C03641=1057.884,320.062,395.291,173.371,36.234,156.810
C03642=1057.890,320.310,395.258,173.375,36.239,156.811
C03643=1057.896,320.558,395.223,173.378,36.243,156.812
C03644=1057.903,320.805,395.190,173.382,36.248,156.813
C03645=1057.909,321.053,395.155,173.385,36.252,156.814
C03646=1057.916,321.300,395.122,173.389,36.256,156.815
C03647=1057.922,321.548,395.087,173.392,36.260,156.816
C03648=1057.930,321.796,395.054,173.396,36.264,156.817
C03649=1057.935,322.043,395.020,173.399,36.269,156.818
C03650=1057.943,322.291,394.986,173.403,36.273,156.819
C03651=1057.949,322.539,394.951,173.406,36.277,156.820
C03652=1057.955,322.786,394.917,173.411,36.281,156.821
C03653=1057.962,323.034,394.883,173.414,36.285,156.822
C03654=1057.969,323.282,394.849,173.418,36.290,156.823
C03655=1057.976,323.528,394.815,173.421,36.294,156.823
C03656=1057.982,323.776,394.780,173.425,36.299,156.824
C03657=1057.988,324.024,394.746,173.429,36.303,156.825
C03658=1057.995,324.271,394.713,173.432,36.307,156.826
C03659=1058.002,324.519,394.678,173.436,36.311,156.827
C03660=1058.009,324.767,394.644,173.439,36.316,156.828
C03661=1058.016,325.014,394.609,173.443,36.320,156.829
C03662=1058.021,325.261,394.575,173.446,36.324,156.830
C03663=1058.029,325.509,394.541,173.451,36.328,156.831
C03664=1058.035,325.757,394.507,173.454,36.333,156.832
C03665=1058.043,326.004,394.472,173.458,36.337,156.833
C03666=1058.049,326.252,394.438,173.461,36.341,156.834
C03667=1058.055,326.499,394.404,173.465,36.345,156.835
C03668=1058.062,326.747,394.370,173.469,36.350,156.836
C03669=1058.069,326.994,394.335,173.472,36.355,156.837
C03670=1058.075,327.242,394.300,173.477,36.359,156.838
C03671=1058.083,327.489,394.266,173.480,36.363,156.839
C03672=1058.089,327.737,394.231,173.484,36.367,156.840
C03673=1058.095,327.985,394.197,173.487,36.372,156.841
C03674=1058.103,328.232,394.163,173.491,36.376,156.842
C03675=1058.109,328.480,394.128,173.494,36.380,156.843
C03676=1058.116,328.727,394.093,173.499,36.385,156.844
C03677=1058.123,328.975,394.060,173.503,36.389,156.845
C03678=1058.130,329.222,394.024,173.506,36.393,156.846
C03679=1058.136,329.470,393.990,173.510,36.398,156.847
C03680=1058.144,329.717,393.955,173.513,36.402,156.848
C03681=1058.150,329.965,393.921,173.518,36.407,156.849
C03682=1058.157,330.212,393.886,173.521,36.411,156.850
C03683=1058.164,330.460,393.852,173.525,36.416,156.851
C03684=1058.170,330.708,393.816,173.529,36.420,156.852
C03685=1058.177,330.955,393.781,173.532,36.424,156.853
C03686=1058.183,331.202,393.747,173.536,36.429,156.854
C03687=1058.190,331.450,393.712,173.540,36.433,156.855
C03688=1058.197,331.702,393.676,173.544,36.438,156.856
C03689=1058.204,331.954,393.641,173.548,36.442,156.857
C03690=1058.210,332.205,393.605,173.551,36.447,156.858
C03691=1058.218,332.457,393.570,173.556,36.452,156.859
C03692=1058.224,332.705,393.535,173.559,36.456,156.860
C03693=1058.231,332.952,393.500,173.563,36.461,156.861
C03694=1058.237,333.200,393.464,173.567,36.465,156.862
C03695=1058.244,333.447,393.429,173.571,36.470,156.863
C03696=1058.250,333.695,393.394,173.575,36.474,156.864
C03697=1058.257,333.943,393.359,173.578,36.479,156.865
C03698=1058.264,334.190,393.324,173.582,36.483,156.866
C03699=1058.271,334.437,393.289,173.587,36.488,156.867
C03700=1058.277,334.685,393.254,173.590,36.493,156.868
C03701=1058.284,334.932,393.219,173.594,36.497,156.869
C03702=1058.291,335.179,393.184,173.598,36.502,156.870
C03703=1058.298,335.427,393.148,173.602,36.507,156.871
C03704=1058.305,335.674,393.113,173.606,36.511,156.872
C03705=1058.311,335.921,393.078,173.609,36.516,156.873
C03706=1058.317,336.169,393.042,173.613,36.520,156.874
C03707=1058.324,336.417,393.007,173.618,36.525,156.876
C03708=1058.331,336.664,392.972,173.621,36.529,156.877
C03709=1058.338,336.911,392.936,173.625,36.534,156.878
C03710=1058.345,337.158,392.901,173.630,36.538,156.879
C03711=1058.351,337.406,392.865,173.633,36.544,156.880
C03712=1058.358,337.654,392.830,173.637,36.548,156.881
C03713=1058.365,337.901,392.795,173.641,36.553,156.882
C03714=1058.371,338.148,392.758,173.645,36.557,156.883
C03715=1058.378,338.396,392.723,173.649,36.562,156.884
C03716=1058.385,338.643,392.688,173.652,36.567,156.885
C03717=1058.392,338.890,392.653,173.657,36.571,156.886
C03718=1058.398,339.137,392.616,173.661,36.576,156.887
C03719=1058.405,339.385,392.581,173.664,36.581,156.888
C03720=1058.412,339.633,392.546,173.669,36.585,156.889
C03721=1058.418,339.880,392.509,173.673,36.591,156.891
C03722=1058.425,340.127,392.474,173.676,36.595,156.892
C03723=1058.431,340.374,392.438,173.681,36.600,156.893
C03724=1058.439,340.622,392.402,173.685,36.605,156.894
C03725=1058.446,340.869,392.366,173.688,36.609,156.895
C03726=1058.452,341.117,392.331,173.693,36.614,156.896
C03727=1058.459,341.364,392.296,173.697,36.619,156.897
C03728=1058.466,341.612,392.259,173.700,36.624,156.898
C03729=1058.473,341.859,392.223,173.705,36.628,156.899
C03730=1058.479,342.106,392.188,173.709,36.633,156.900
C03731=1058.487,342.353,392.152,173.713,36.638,156.901
C03732=1058.493,342.601,392.116,173.717,36.643,156.903
C03733=1058.500,342.848,392.080,173.721,36.648,156.904
C03734=1058.506,343.095,392.044,173.725,36.652,156.905
C03735=1058.514,343.343,392.008,173.729,36.657,156.906
C03736=1058.520,343.590,391.972,173.734,36.662,156.907
C03737=1058.527,343.837,391.936,173.738,36.667,156.908
C03738=1058.534,344.085,391.900,173.741,36.672,156.909
C03739=1058.541,344.332,391.864,173.746,36.677,156.910
C03740=1058.547,344.579,391.827,173.750,36.681,156.912
C03741=1058.554,344.827,391.791,173.754,36.686,156.913
C03742=1058.561,345.074,391.755,173.758,36.692,156.914
C03743=1058.567,345.321,391.719,173.762,36.696,156.915
C03744=1058.574,345.569,391.682,173.766,36.701,156.916
C03745=1058.581,345.816,391.646,173.770,36.706,156.917
C03746=1058.588,346.064,391.610,173.775,36.711,156.918
C03747=1058.594,346.311,391.574,173.779,36.716,156.919
C03748=1058.602,346.558,391.538,173.783,36.721,156.921
C03749=1058.608,346.805,391.501,173.787,36.726,156.922
C03750=1058.615,347.053,391.464,173.792,36.731,156.923
C03751=1058.622,347.300,391.428,173.796,36.736,156.924
C03752=1058.629,347.548,391.392,173.800,36.741,156.925
C03753=1058.636,347.795,391.355,173.804,36.746,156.927
C03754=1058.643,348.042,391.319,173.809,36.751,156.928
C03755=1058.650,348.289,391.283,173.812,36.756,156.929
C03756=1058.656,348.536,391.246,173.816,36.761,156.930
C03757=1058.663,348.784,391.209,173.821,36.766,156.931
C03758=1058.670,349.030,391.173,173.825,36.771,156.932
C03759=1058.677,349.278,391.136,173.829,36.776,156.933
C03760=1058.684,349.525,391.099,173.833,36.781,156.935
C03761=1058.691,349.773,391.063,173.838,36.786,156.936
C03762=1058.698,350.020,391.027,173.843,36.791,156.937
C03763=1058.705,350.267,390.989,173.846,36.796,156.938
C03764=1058.712,350.514,390.952,173.851,36.801,156.939
C03765=1058.718,350.762,390.916,173.855,36.806,156.941
C03766=1058.726,351.009,390.880,173.860,36.811,156.942
C03767=1058.733,351.255,390.843,173.863,36.816,156.943
C03768=1058.739,351.503,390.806,173.868,36.822,156.944
C03769=1058.746,351.750,390.769,173.872,36.827,156.945
C03770=1058.753,351.997,390.732,173.877,36.832,156.947
C03771=1058.760,352.245,390.695,173.881,36.837,156.948
C03772=1058.767,352.492,390.658,173.885,36.842,156.949
C03773=1058.774,352.739,390.621,173.889,36.848,156.950
C03774=1058.780,352.986,390.584,173.894,36.853,156.951
C03775=1058.787,353.233,390.547,173.899,36.858,156.953
C03776=1058.794,353.481,390.510,173.903,36.863,156.954
C03777=1058.801,353.728,390.473,173.907,36.868,156.955
C03778=1058.808,353.975,390.436,173.911,36.873,156.956
C03779=1058.815,354.222,390.398,173.916,36.879,156.958
C03780=1058.822,354.469,390.362,173.921,36.884,156.959
C03781=1058.829,354.716,390.324,173.924,36.889,156.960
C03782=1058.836,354.963,390.287,173.929,36.895,156.961
C03783=1058.842,355.210,390.250,173.933,36.900,156.963
C03784=1058.850,355.457,390.213,173.938,36.905,156.964
C03785=1058.857,355.705,390.175,173.943,36.910,156.965
C03786=1058.863,355.952,390.139,173.947,36.916,156.966
C03787=1058.870,356.199,390.101,173.951,36.921,156.968
C03788=1058.878,356.446,390.064,173.955,36.926,156.969
C03789=1058.885,356.693,390.026,173.960,36.931,156.970
C03790=1058.892,356.939,389.989,173.965,36.937,156.971
C03791=1058.899,357.187,389.951,173.969,36.942,156.973
C03792=1058.906,357.434,389.915,173.973,36.947,156.974
C03793=1058.913,357.681,389.877,173.978,36.952,156.975
C03794=1058.920,357.929,389.839,173.982,36.958,156.976
C03795=1058.927,358.176,389.802,173.987,36.964,156.978
C03796=1058.934,358.422,389.765,173.992,36.969,156.979
C03797=1058.941,358.669,389.727,173.996,36.974,156.980
C03798=1058.948,358.917,389.689,174.001,36.980,156.982
C03799=1058.955,359.164,389.652,174.005,36.985,156.983
C03800=1058.963,359.416,389.613,174.010,36.991,156.984
C03801=1058.970,359.668,389.575,174.014,36.996,156.986
C03802=1058.976,359.920,389.536,174.019,37.002,156.987
C03803=1058.983,360.172,389.498,174.024,37.008,156.988
C03804=1058.991,360.419,389.460,174.029,37.013,156.990
C03805=1058.998,360.666,389.422,174.033,37.019,156.991
C03806=1059.005,360.913,389.384,174.038,37.024,156.992
C03807=1059.012,361.160,389.346,174.042,37.029,156.993
C03808=1059.019,361.408,389.309,174.047,37.035,156.995
C03809=1059.026,361.655,389.271,174.051,37.040,156.996
C03810=1059.033,361.902,389.233,174.056,37.046,156.997
C03811=1059.040,362.149,389.195,174.061,37.051,156.999
C03812=1059.048,362.396,389.157,174.066,37.057,157.000
C03813=1059.054,362.643,389.119,174.070,37.062,157.001
C03814=1059.062,362.890,389.081,174.075,37.068,157.003
C03815=1059.069,363.136,389.043,174.080,37.074,157.004
C03816=1059.076,363.384,389.005,174.085,37.080,157.005
C03817=1059.083,363.631,388.967,174.088,37.085,157.007
C03818=1059.091,363.877,388.929,174.093,37.091,157.008
C03819=1059.097,364.125,388.891,174.098,37.096,157.009
C03820=1059.105,364.371,388.853,174.103,37.102,157.011
C03821=1059.111,364.618,388.814,174.107,37.108,157.012
C03822=1059.119,364.865,388.776,174.112,37.113,157.014
C03823=1059.125,365.112,388.737,174.117,37.119,157.015
C03824=1059.132,365.359,388.699,174.122,37.125,157.016
C03825=1059.140,365.606,388.661,174.127,37.131,157.018
C03826=1059.146,365.853,388.622,174.131,37.137,157.019
C03827=1059.154,366.099,388.584,174.136,37.142,157.021
C03828=1059.160,366.347,388.546,174.141,37.148,157.022
C03829=1059.168,366.593,388.508,174.146,37.154,157.023
C03830=1059.175,366.840,388.469,174.151,37.159,157.025
C03831=1059.182,367.087,388.430,174.156,37.165,157.026
C03832=1059.190,367.334,388.391,174.160,37.171,157.027
C03833=1059.197,367.581,388.352,174.165,37.177,157.029
C03834=1059.204,367.828,388.315,174.170,37.183,157.030
C03835=1059.211,368.075,388.276,174.175,37.189,157.032
C03836=1059.217,368.322,388.237,174.180,37.195,157.033
C03837=1059.225,368.568,388.199,174.184,37.200,157.035
C03838=1059.232,368.816,388.160,174.189,37.206,157.036
C03839=1059.240,369.062,388.122,174.194,37.212,157.038
C03840=1059.247,369.309,388.083,174.199,37.218,157.039
C03841=1059.254,369.556,388.044,174.203,37.224,157.040
C03842=1059.261,369.803,388.006,174.208,37.230,157.042
C03843=1059.269,370.050,387.966,174.214,37.236,157.043
C03844=1059.276,370.296,387.927,174.218,37.241,157.045
C03845=1059.283,370.543,387.889,174.223,37.247,157.046
C03846=1059.291,370.790,387.849,174.229,37.254,157.048
C03847=1059.298,371.037,387.811,174.234,37.260,157.049
C03848=1059.305,371.284,387.772,174.239,37.266,157.051
C03849=1059.312,371.531,387.733,174.244,37.272,157.052
C03850=1059.320,371.777,387.694,174.249,37.278,157.053
C03851=1059.327,372.024,387.655,174.254,37.283,157.055
C03852=1059.334,372.271,387.616,174.259,37.289,157.056
C03853=1059.342,372.518,387.577,174.264,37.296,157.058
C03854=1059.348,372.765,387.538,174.269,37.302,157.059
C03855=1059.356,373.012,387.499,174.274,37.308,157.061
C03856=1059.364,373.282,387.455,174.279,37.314,157.062
C03857=1059.372,373.553,387.413,174.284,37.321,157.064
C03858=1059.380,373.823,387.369,174.290,37.328,157.066
C03859=1059.388,374.094,387.327,174.296,37.335,157.067
C03860=1059.395,374.340,387.287,174.301,37.341,157.069
C03861=1059.403,374.587,387.247,174.306,37.347,157.071
C03862=1059.409,374.834,387.209,174.311,37.353,157.072
C03863=1059.417,375.081,387.169,174.316,37.359,157.074
C03864=1059.424,375.327,387.129,174.321,37.366,157.075
C03865=1059.431,375.574,387.090,174.326,37.372,157.077
C03866=1059.439,375.820,387.050,174.331,37.379,157.078
C03867=1059.446,376.067,387.011,174.336,37.385,157.080
C03868=1059.453,376.314,386.972,174.341,37.391,157.081
C03869=1059.460,376.560,386.932,174.347,37.397,157.083
C03870=1059.468,376.807,386.892,174.352,37.404,157.084
C03871=1059.475,377.053,386.853,174.358,37.410,157.086
C03872=1059.483,377.300,386.813,174.363,37.416,157.088
C03873=1059.490,377.547,386.773,174.368,37.422,157.089
C03874=1059.498,377.794,386.734,174.373,37.429,157.091
C03875=1059.505,378.041,386.694,174.378,37.435,157.092
C03876=1059.512,378.287,386.654,174.383,37.441,157.094
C03877=1059.520,378.534,386.614,174.389,37.448,157.095
C03878=1059.527,378.780,386.575,174.394,37.455,157.097
C03879=1059.535,379.027,386.535,174.399,37.461,157.099
C03880=1059.543,379.274,386.495,174.404,37.467,157.100
C03881=1059.550,379.520,386.456,174.410,37.474,157.102
C03882=1059.558,379.767,386.415,174.415,37.480,157.103
C03883=1059.566,380.014,386.375,174.421,37.487,157.105
C03884=1059.572,380.260,386.335,174.426,37.493,157.107
C03885=1059.580,380.507,386.295,174.431,37.499,157.108
C03886=1059.587,380.754,386.255,174.436,37.506,157.110
C03887=1059.595,381.001,386.215,174.442,37.513,157.112
C03888=1059.603,381.246,386.175,174.448,37.519,157.113
C03889=1059.610,381.494,386.134,174.453,37.526,157.115
C03890=1059.617,381.740,386.095,174.458,37.532,157.116
C03891=1059.624,381.986,386.054,174.463,37.539,157.118
C03892=1059.632,382.233,386.014,174.469,37.546,157.120
C03893=1059.640,382.480,385.973,174.475,37.553,157.122
C03894=1059.646,382.726,385.933,174.480,37.559,157.123
C03895=1059.654,382.972,385.892,174.485,37.566,157.125
C03896=1059.662,383.219,385.852,174.490,37.573,157.127
C03897=1059.669,383.466,385.811,174.496,37.579,157.128
C03898=1059.676,383.712,385.771,174.502,37.586,157.130
C03899=1059.684,383.958,385.731,174.507,37.593,157.132
C03900=1059.691,384.206,385.690,174.512,37.599,157.133
C03901=1059.699,384.452,385.650,174.518,37.606,157.135
C03902=1059.707,384.698,385.608,174.524,37.613,157.137
C03903=1059.714,384.945,385.569,174.529,37.620,157.138
C03904=1059.722,385.191,385.528,174.535,37.627,157.140
C03905=1059.729,385.438,385.487,174.541,37.633,157.142
C03906=1059.737,385.684,385.446,174.546,37.640,157.144
C03907=1059.744,385.931,385.406,174.552,37.648,157.145
C03908=1059.752,386.177,385.365,174.557,37.654,157.147
C03909=1059.760,386.424,385.325,174.563,37.661,157.149
C03910=1059.767,386.670,385.283,174.568,37.668,157.151
C03911=1059.775,386.916,385.243,174.574,37.675,157.152
C03912=1059.782,387.156,385.203,174.580,37.682,157.154
C03913=1059.790,387.396,385.163,174.585,37.688,157.156
C03914=1059.797,387.636,385.123,174.591,37.695,157.157
C03915=1059.805,387.874,385.084,174.596,37.702,157.159
C03916=1059.813,388.115,385.044,174.602,37.709,157.161
C03917=1059.820,388.353,385.004,174.608,37.716,157.163
C03918=1059.827,388.594,384.964,174.613,37.722,157.164
C03919=1059.835,388.833,384.925,174.618,37.729,157.166
C03920=1059.843,389.079,384.883,174.625,37.736,157.168
C03921=1059.851,389.326,384.842,174.630,37.743,157.170
C03922=1059.858,389.572,384.801,174.636,37.750,157.171
C03923=1059.866,389.819,384.760,174.642,37.757,157.173
C03924=1059.874,390.065,384.719,174.647,37.765,157.175
C03925=1059.882,390.312,384.677,174.653,37.772,157.177
C03926=1059.890,390.558,384.636,174.659,37.779,157.179
C03927=1059.897,390.805,384.595,174.665,37.786,157.181
C03928=1059.905,391.051,384.553,174.671,37.793,157.182
C03929=1059.913,391.297,384.512,174.677,37.801,157.184
C03930=1059.920,391.543,384.470,174.683,37.808,157.186
C03931=1059.928,391.790,384.429,174.689,37.815,157.188
C03932=1059.936,392.036,384.387,174.694,37.822,157.190
C03933=1059.944,392.283,384.346,174.700,37.830,157.192
C03934=1059.951,392.529,384.304,174.706,37.837,157.194
C03935=1059.959,392.775,384.263,174.712,37.844,157.196
C03936=1059.968,393.021,384.221,174.718,37.852,157.197
C03937=1059.975,393.267,384.179,174.724,37.859,157.199
C03938=1059.983,393.513,384.138,174.730,37.866,157.201
C03939=1059.990,393.760,384.096,174.736,37.874,157.203
C03940=1059.998,394.007,384.054,174.742,37.881,157.205
C03941=1060.006,394.253,384.012,174.749,37.889,157.207
C03942=1060.014,394.499,383.970,174.754,37.897,157.209
C03943=1060.021,394.746,383.928,174.761,37.904,157.211
C03944=1060.029,394.992,383.887,174.766,37.912,157.213
C03945=1060.037,395.238,383.845,174.773,37.919,157.215
C03946=1060.046,395.484,383.803,174.778,37.927,157.217
C03947=1060.053,395.730,383.761,174.785,37.934,157.219
C03948=1060.061,395.976,383.719,174.790,37.942,157.221
C03949=1060.069,396.223,383.677,174.797,37.950,157.223
C03950=1060.076,396.469,383.635,174.804,37.957,157.225
C03951=1060.085,396.716,383.592,174.809,37.965,157.227
C03952=1060.092,396.961,383.550,174.816,37.972,157.228
C03953=1060.100,397.208,383.508,174.822,37.980,157.231
C03954=1060.108,397.453,383.466,174.828,37.988,157.232
C03955=1060.117,397.700,383.423,174.835,37.996,157.235
C03956=1060.127,398.015,383.369,174.843,38.005,157.237
C03957=1060.136,398.330,383.315,174.851,38.015,157.240
C03958=1060.147,398.646,383.261,174.859,38.025,157.242
C03959=1060.157,398.960,383.206,174.867,38.036,157.245
C03960=1060.165,399.207,383.163,174.872,38.043,157.247
C03961=1060.172,399.453,383.121,174.879,38.051,157.249
C03962=1060.181,399.699,383.078,174.886,38.059,157.251
C03963=1060.189,399.946,383.036,174.891,38.067,157.253
C03964=1060.197,400.192,382.993,174.898,38.075,157.255
C03965=1060.205,400.438,382.951,174.905,38.083,157.257
C03966=1060.213,400.685,382.907,174.912,38.091,157.260
C03967=1060.220,400.931,382.865,174.917,38.099,157.262
C03968=1060.231,401.250,382.810,174.926,38.109,157.264
C03969=1060.242,401.569,382.754,174.935,38.120,157.267
C03970=1060.253,401.887,382.699,174.943,38.130,157.270
C03971=1060.264,402.206,382.643,174.951,38.141,157.273
C03972=1060.271,402.452,382.600,174.958,38.149,157.275
C03973=1060.280,402.699,382.557,174.965,38.157,157.277
C03974=1060.287,402.944,382.515,174.971,38.165,157.279
C03975=1060.295,403.191,382.471,174.977,38.174,157.281
C03976=1060.304,403.437,382.428,174.984,38.181,157.283
C03977=1060.312,403.683,382.385,174.991,38.190,157.286
C03978=1060.320,403.929,382.341,174.997,38.198,157.288
C03979=1060.328,404.175,382.298,175.004,38.206,157.290
C03980=1060.336,404.421,382.255,175.011,38.215,157.292
C03981=1060.345,404.668,382.212,175.017,38.223,157.294
C03982=1060.352,404.913,382.168,175.024,38.231,157.296
C03983=1060.360,405.159,382.125,175.031,38.240,157.299
C03984=1060.368,405.405,382.081,175.037,38.248,157.301
C03985=1060.377,405.651,382.038,175.044,38.257,157.303
C03986=1060.385,405.897,381.994,175.051,38.265,157.305
C03987=1060.393,406.143,381.951,175.058,38.274,157.308
C03988=1060.401,406.389,381.907,175.065,38.282,157.310
C03989=1060.409,406.636,381.863,175.072,38.291,157.312
C03990=1060.418,406.882,381.820,175.079,38.299,157.314
C03991=1060.426,407.127,381.776,175.086,38.308,157.317
C03992=1060.435,407.374,381.733,175.093,38.317,157.319
C03993=1060.443,407.620,381.688,175.099,38.325,157.321
C03994=1060.451,407.866,381.645,175.106,38.333,157.324
C03995=1060.459,408.112,381.601,175.113,38.342,157.326
C03996=1060.467,408.358,381.557,175.120,38.351,157.328
C03997=1060.475,408.604,381.513,175.127,38.360,157.331
C03998=1060.484,408.849,381.469,175.134,38.369,157.333
C03999=1060.492,409.096,381.425,175.141,38.377,157.335
C04000=1060.500,409.342,381.381,175.148,38.386,157.338
C04001=1060.509,409.587,381.337,175.155,38.395,157.340
C04002=1060.517,409.833,381.293,175.162,38.404,157.342
C04003=1060.525,410.079,381.248,175.169,38.413,157.345
C04004=1060.534,410.326,381.204,175.176,38.421,157.347
C04005=1060.543,410.571,381.161,175.184,38.430,157.350
C04006=1060.551,410.817,381.116,175.191,38.439,157.352
C04007=1060.559,411.064,381.072,175.198,38.448,157.354
C04008=1060.568,411.309,381.028,175.205,38.457,157.357
C04009=1060.576,411.555,380.984,175.213,38.466,157.359
C04010=1060.585,411.801,380.939,175.220,38.475,157.362
C04011=1060.593,412.047,380.895,175.228,38.484,157.364
C04012=1060.602,412.293,380.850,175.235,38.493,157.367
C04013=1060.611,412.538,380.805,175.242,38.502,157.369
C04014=1060.619,412.785,380.761,175.249,38.511,157.372
C04015=1060.627,413.030,380.716,175.257,38.520,157.374
C04016=1060.637,413.277,380.672,175.264,38.530,157.377
C04017=1060.645,413.522,380.628,175.271,38.538,157.379
C04018=1060.654,413.768,380.582,175.279,38.548,157.382
C04019=1060.662,414.014,380.538,175.287,38.557,157.384
C04020=1060.671,414.260,380.493,175.294,38.566,157.387
C04021=1060.679,414.505,380.448,175.301,38.576,157.389
C04022=1060.688,414.751,380.403,175.309,38.585,157.392
C04023=1060.696,414.997,380.359,175.317,38.594,157.394
C04024=1060.708,415.321,380.299,175.327,38.607,157.398
C04025=1060.719,415.646,380.240,175.337,38.620,157.401
C04026=1060.730,415.969,380.180,175.347,38.632,157.404
C04027=1060.742,416.294,380.120,175.357,38.645,157.408
C04028=1060.750,416.540,380.076,175.365,38.654,157.411
C04029=1060.759,416.785,380.031,175.372,38.663,157.413
C04030=1060.768,417.031,379.985,175.380,38.673,157.416
C04031=1060.776,417.277,379.940,175.388,38.683,157.418
C04032=1060.785,417.522,379.894,175.395,38.693,157.421
C04033=1060.794,417.768,379.849,175.403,38.702,157.424
C04034=1060.803,418.014,379.803,175.411,38.712,157.426
C04035=1060.811,418.259,379.758,175.419,38.721,157.429
C04036=1060.820,418.505,379.713,175.427,38.731,157.432
C04037=1060.829,418.751,379.667,175.435,38.741,157.434
C04038=1060.838,418.997,379.622,175.443,38.751,157.437
C04039=1060.846,419.243,379.576,175.451,38.761,157.440
C04040=1060.856,419.488,379.530,175.459,38.771,157.443
C04041=1060.865,419.734,379.484,175.467,38.780,157.445
C04042=1060.874,419.980,379.439,175.475,38.790,157.448
C04043=1060.882,420.225,379.394,175.484,38.800,157.451
C04044=1060.891,420.470,379.348,175.491,38.810,157.454
C04045=1060.900,420.716,379.302,175.499,38.820,157.456
C04046=1060.909,420.961,379.256,175.507,38.830,157.459
C04047=1060.917,421.207,379.210,175.515,38.840,157.462
C04048=1060.926,421.453,379.164,175.524,38.850,157.465
C04049=1060.936,421.698,379.117,175.532,38.860,157.468
C04050=1060.944,421.944,379.071,175.540,38.871,157.471
C04051=1060.953,422.189,379.025,175.549,38.881,157.473
C04052=1060.962,422.435,378.979,175.557,38.891,157.476
C04053=1060.971,422.681,378.933,175.565,38.901,157.479
C04054=1060.979,422.926,378.886,175.573,38.911,157.482
C04055=1060.989,423.172,378.840,175.582,38.922,157.485
C04056=1060.998,423.417,378.794,175.591,38.932,157.488
C04057=1061.007,423.663,378.747,175.598,38.942,157.491
C04058=1061.016,423.908,378.701,175.607,38.953,157.494
C04059=1061.025,424.153,378.654,175.616,38.964,157.497
C04060=1061.034,424.399,378.608,175.624,38.974,157.500
C04061=1061.043,424.645,378.561,175.633,38.984,157.502
C04062=1061.052,424.890,378.515,175.642,38.995,157.505
C04063=1061.061,425.136,378.468,175.651,39.005,157.508
C04064=1061.071,425.381,378.422,175.658,39.016,157.511
C04065=1061.080,425.626,378.374,175.667,39.026,157.514
C04066=1061.089,425.872,378.328,175.676,39.037,157.517
C04067=1061.098,426.118,378.281,175.685,39.048,157.520
C04068=1061.108,426.362,378.234,175.693,39.058,157.523
C04069=1061.116,426.608,378.187,175.702,39.069,157.526
C04070=1061.126,426.854,378.141,175.711,39.080,157.530
C04071=1061.135,427.099,378.093,175.720,39.091,157.533
C04072=1061.145,427.344,378.046,175.729,39.102,157.536
C04073=1061.154,427.589,377.999,175.738,39.113,157.539
C04074=1061.163,427.834,377.952,175.747,39.123,157.542
C04075=1061.172,428.080,377.904,175.755,39.134,157.545
C04076=1061.181,428.325,377.857,175.765,39.145,157.548
C04077=1061.191,428.571,377.810,175.774,39.156,157.551
C04078=1061.200,428.816,377.763,175.783,39.167,157.555
C04079=1061.209,429.061,377.715,175.792,39.179,157.558
C04080=1061.222,429.406,377.648,175.805,39.194,157.562
C04081=1061.236,429.750,377.582,175.818,39.210,157.567
C04082=1061.249,430.095,377.515,175.831,39.226,157.571
C04083=1061.262,430.440,377.448,175.844,39.242,157.576
C04084=1061.272,430.686,377.400,175.853,39.253,157.579
C04085=1061.281,430.931,377.352,175.862,39.264,157.582
C04086=1061.290,431.176,377.304,175.872,39.275,157.586
C04087=1061.300,431.421,377.256,175.882,39.287,157.589
C04088=1061.309,431.667,377.209,175.891,39.298,157.592
C04089=1061.318,431.911,377.160,175.900,39.310,157.596
C04090=1061.328,432.157,377.113,175.910,39.322,157.599
C04091=1061.337,432.402,377.064,175.919,39.333,157.602
C04092=1061.347,432.647,377.016,175.929,39.344,157.606
C04093=1061.357,432.892,376.968,175.939,39.356,157.609
C04094=1061.366,433.137,376.920,175.948,39.368,157.612
C04095=1061.375,433.382,376.872,175.958,39.379,157.616
C04096=1061.385,433.627,376.823,175.968,39.391,157.619
C04097=1061.395,433.872,376.775,175.978,39.403,157.623
C04098=1061.404,434.118,376.727,175.987,39.415,157.626
C04099=1061.414,434.362,376.678,175.998,39.427,157.630
C04100=1061.424,434.607,376.630,176.007,39.438,157.633
C04101=1061.434,434.852,376.581,176.017,39.450,157.637
C04102=1061.443,435.097,376.533,176.027,39.463,157.640
C04103=1061.453,435.342,376.484,176.037,39.474,157.644
C04104=1061.463,435.587,376.436,176.047,39.486,157.647
C04105=1061.473,435.832,376.387,176.057,39.498,157.651
C04106=1061.482,436.077,376.337,176.067,39.511,157.654
C04107=1061.492,436.323,376.289,176.077,39.523,157.658
C04108=1061.502,436.568,376.240,176.087,39.535,157.661
C04109=1061.512,436.813,376.192,176.098,39.547,157.665
C04110=1061.522,437.057,376.142,176.107,39.559,157.669
C04111=1061.532,437.302,376.094,176.118,39.571,157.672
C04112=1061.542,437.547,376.044,176.129,39.584,157.676
C04113=1061.552,437.792,375.996,176.139,39.596,157.679
C04114=1061.561,438.037,375.946,176.149,39.608,157.683
C04115=1061.572,438.282,375.897,176.160,39.621,157.687
C04116=1061.582,438.527,375.848,176.170,39.633,157.691
C04117=1061.591,438.771,375.798,176.181,39.646,157.694
C04118=1061.602,439.016,375.748,176.192,39.659,157.698
C04119=1061.612,439.261,375.700,176.201,39.671,157.702
C04120=1061.621,439.506,375.650,176.212,39.684,157.706
C04121=1061.632,439.751,375.600,176.223,39.696,157.709
C04122=1061.642,439.995,375.551,176.234,39.709,157.713
C04123=1061.652,440.241,375.501,176.244,39.722,157.717
C04124=1061.662,440.485,375.452,176.255,39.735,157.721
C04125=1061.672,440.730,375.401,176.266,39.747,157.725
C04126=1061.682,440.974,375.351,176.277,39.760,157.729
C04127=1061.692,441.220,375.301,176.288,39.773,157.733
C04128=1061.702,441.464,375.252,176.299,39.786,157.736
C04129=1061.713,441.708,375.202,176.310,39.799,157.740
C04130=1061.723,441.954,375.151,176.321,39.812,157.744
C04131=1061.733,442.198,375.102,176.333,39.825,157.748
C04132=1061.743,442.443,375.051,176.344,39.839,157.752
C04133=1061.754,442.687,375.001,176.355,39.852,157.756
C04134=1061.764,442.933,374.951,176.366,39.865,157.760
C04135=1061.774,443.177,374.900,176.377,39.878,157.764
C04136=1061.784,443.408,374.853,176.388,39.891,157.768
C04137=1061.794,443.637,374.805,176.399,39.903,157.772
C04138=1061.803,443.868,374.758,176.409,39.916,157.776
C04139=1061.813,444.098,374.710,176.420,39.929,157.780
C04140=1061.822,444.328,374.663,176.431,39.941,157.784
C04141=1061.832,444.559,374.614,176.441,39.954,157.787
C04142=1061.843,444.789,374.568,176.452,39.967,157.791
C04143=1061.853,445.020,374.519,176.463,39.980,157.795
C04144=1061.862,445.264,374.469,176.476,39.993,157.799
C04145=1061.873,445.509,374.418,176.487,40.007,157.804
C04146=1061.884,445.753,374.367,176.499,40.021,157.808
C04147=1061.895,445.998,374.316,176.511,40.034,157.812
C04148=1061.905,446.243,374.265,176.523,40.048,157.816
C04149=1061.916,446.487,374.214,176.534,40.062,157.821
C04150=1061.926,446.731,374.163,176.547,40.076,157.825
C04151=1061.937,446.975,374.111,176.558,40.090,157.829
C04152=1061.948,447.218,374.060,176.571,40.104,157.834
C04153=1061.958,447.462,374.010,176.583,40.118,157.838
C04154=1061.970,447.705,373.959,176.595,40.132,157.842
C04155=1061.983,447.950,373.909,176.607,40.145,157.846
C04156=1061.997,448.194,373.860,176.619,40.158,157.851
C04157=1062.011,448.438,373.812,176.632,40.171,157.855
C04158=1062.027,448.682,373.764,176.645,40.184,157.859
C04159=1062.044,448.928,373.717,176.657,40.196,157.863
C04160=1062.060,449.172,373.670,176.670,40.208,157.867
C04161=1062.079,449.418,373.624,176.683,40.220,157.870
C04162=1062.098,449.662,373.579,176.696,40.232,157.874
C04163=1062.118,449.908,373.535,176.709,40.243,157.878
C04164=1061.785,449.918,373.260,176.702,40.360,157.910
C04165=1061.764,449.672,373.305,176.689,40.349,157.906
C04166=1061.745,449.427,373.350,176.676,40.338,157.902
C04167=1061.726,449.182,373.396,176.663,40.326,157.899
C04168=1061.708,448.937,373.443,176.650,40.314,157.895
C04169=1061.693,448.692,373.490,176.638,40.301,157.891
C04170=1061.677,448.448,373.538,176.625,40.289,157.887
C04171=1061.662,448.202,373.586,176.612,40.276,157.883
C04172=1061.648,447.960,373.635,176.600,40.263,157.879
C04173=1061.635,447.715,373.685,176.587,40.249,157.874
C04174=1061.623,447.471,373.736,176.575,40.236,157.870
C04175=1061.612,447.228,373.786,176.563,40.222,157.866
C04176=1061.601,446.985,373.837,176.551,40.208,157.861
C04177=1061.591,446.741,373.889,176.539,40.194,157.857
C04178=1061.580,446.496,373.939,176.527,40.181,157.853
C04179=1061.569,446.251,373.991,176.514,40.167,157.848
C04180=1061.559,446.007,374.042,176.503,40.153,157.844
C04181=1061.548,445.762,374.092,176.490,40.139,157.840
C04182=1061.537,445.518,374.144,176.479,40.126,157.836
C04183=1061.527,445.273,374.195,176.467,40.112,157.831
C04184=1061.516,445.029,374.245,176.455,40.099,157.827
C04185=1061.507,444.808,374.291,176.444,40.086,157.824
C04186=1061.497,444.588,374.337,176.434,40.074,157.820
C04187=1061.488,444.367,374.383,176.424,40.062,157.816
C04188=1061.478,444.146,374.429,176.413,40.050,157.812
C04189=1061.469,443.926,374.474,176.403,40.038,157.809
C04190=1061.460,443.705,374.520,176.392,40.026,157.805
C04191=1061.451,443.484,374.566,176.382,40.013,157.801
C04192=1061.441,443.264,374.610,176.372,40.001,157.797
C04193=1061.431,443.019,374.661,176.361,39.988,157.794
C04194=1061.421,442.774,374.712,176.348,39.975,157.789
C04195=1061.410,442.529,374.762,176.337,39.962,157.785
C04196=1061.399,442.285,374.813,176.326,39.949,157.781
C04197=1061.389,442.040,374.862,176.315,39.936,157.777
C04198=1061.379,441.796,374.913,176.304,39.923,157.773
C04199=1061.368,441.551,374.963,176.293,39.910,157.770
C04200=1061.358,441.307,375.013,176.282,39.897,157.766
C04201=1061.348,441.061,375.063,176.271,39.884,157.762
C04202=1061.337,440.816,375.112,176.259,39.871,157.758
C04203=1061.328,440.572,375.162,176.248,39.858,157.754
C04204=1061.317,440.327,375.212,176.237,39.845,157.750
C04205=1061.308,440.083,375.262,176.227,39.833,157.746
C04206=1061.297,439.838,375.312,176.216,39.820,157.742
C04207=1061.287,439.593,375.361,176.206,39.807,157.739
C04208=1061.277,439.348,375.411,176.195,39.795,157.735
C04209=1061.267,439.104,375.461,176.184,39.782,157.731
C04210=1061.257,438.859,375.509,176.173,39.770,157.727
C04211=1061.247,438.613,375.559,176.163,39.757,157.723
C04212=1061.237,438.369,375.609,176.152,39.745,157.720
C04213=1061.227,438.125,375.658,176.141,39.732,157.716
C04214=1061.218,437.879,375.707,176.131,39.720,157.712
C04215=1061.208,437.634,375.757,176.121,39.707,157.709
C04216=1061.198,437.390,375.806,176.110,39.695,157.705
C04217=1061.187,437.144,375.855,176.100,39.683,157.701
C04218=1061.177,436.900,375.904,176.089,39.671,157.698
C04219=1061.167,436.655,375.952,176.079,39.659,157.694
C04220=1061.158,436.410,376.001,176.069,39.647,157.690
C04221=1061.148,436.165,376.051,176.058,39.634,157.687
C04222=1061.138,435.920,376.100,176.049,39.622,157.683
C04223=1061.128,435.675,376.148,176.038,39.610,157.680
C04224=1061.118,435.430,376.197,176.028,39.598,157.676
C04225=1061.109,435.185,376.245,176.018,39.587,157.673
C04226=1061.099,434.940,376.294,176.008,39.574,157.669
C04227=1061.089,434.695,376.342,175.998,39.563,157.666
C04228=1061.079,434.450,376.391,175.988,39.551,157.662
C04229=1061.070,434.205,376.439,175.979,39.539,157.659
C04230=1061.060,433.960,376.488,175.968,39.527,157.655
C04231=1061.050,433.715,376.536,175.959,39.516,157.652
C04232=1061.040,433.470,376.585,175.948,39.504,157.648
C04233=1061.031,433.225,376.634,175.939,39.492,157.645
C04234=1061.021,432.979,376.681,175.929,39.480,157.641
C04235=1061.011,432.734,376.730,175.920,39.469,157.638
C04236=1061.002,432.489,376.778,175.909,39.457,157.635
C04237=1060.992,432.244,376.826,175.900,39.446,157.631
C04238=1060.983,431.999,376.874,175.891,39.434,157.628
C04239=1060.973,431.754,376.922,175.881,39.423,157.625
C04240=1060.964,431.509,376.971,175.871,39.411,157.621
C04241=1060.954,431.263,377.018,175.862,39.400,157.618
C04242=1060.945,431.018,377.066,175.852,39.389,157.615
C04243=1060.936,430.773,377.114,175.843,39.377,157.611
C04244=1060.926,430.528,377.162,175.834,39.366,157.608
C04245=1060.913,430.182,377.230,175.820,39.350,157.604
C04246=1060.899,429.834,377.296,175.807,39.334,157.599
C04247=1060.886,429.488,377.364,175.794,39.318,157.594
C04248=1060.872,429.141,377.431,175.781,39.303,157.590
C04249=1060.863,428.896,377.479,175.772,39.292,157.587
C04250=1060.854,428.650,377.526,175.762,39.281,157.583
C04251=1060.845,428.405,377.573,175.753,39.270,157.580
C04252=1060.835,428.160,377.621,175.744,39.259,157.577
C04253=1060.826,427.915,377.668,175.735,39.248,157.574
C04254=1060.817,427.669,377.716,175.726,39.237,157.571
C04255=1060.808,427.424,377.763,175.718,39.226,157.568
C04256=1060.798,427.179,377.810,175.709,39.216,157.565
C04257=1060.789,426.934,377.857,175.700,39.204,157.562
C04258=1060.780,426.687,377.904,175.691,39.194,157.558
C04259=1060.771,426.443,377.951,175.682,39.183,157.556
C04260=1060.762,426.197,377.998,175.673,39.173,157.552
C04261=1060.752,425.951,378.044,175.664,39.162,157.549
C04262=1060.743,425.707,378.092,175.655,39.151,157.546
C04263=1060.733,425.461,378.138,175.647,39.141,157.543
C04264=1060.725,425.215,378.185,175.638,39.130,157.540
C04265=1060.716,424.970,378.231,175.629,39.120,157.537
C04266=1060.706,424.724,378.279,175.620,39.109,157.534
C04267=1060.697,424.479,378.325,175.611,39.099,157.531
C04268=1060.688,424.234,378.372,175.603,39.088,157.528
C04269=1060.679,423.988,378.418,175.595,39.078,157.526
C04270=1060.669,423.743,378.465,175.586,39.068,157.523
C04271=1060.661,423.497,378.511,175.578,39.057,157.520
C04272=1060.651,423.252,378.557,175.569,39.047,157.517
C04273=1060.643,423.006,378.604,175.560,39.037,157.514
C04274=1060.633,422.761,378.650,175.553,39.026,157.511
C04275=1060.625,422.516,378.697,175.544,39.016,157.508
C04276=1060.616,422.270,378.742,175.535,39.006,157.505
C04277=1060.607,422.025,378.789,175.527,38.995,157.502
C04278=1060.597,421.778,378.836,175.519,38.986,157.500
C04279=1060.588,421.533,378.881,175.510,38.975,157.497
C04280=1060.580,421.287,378.928,175.502,38.965,157.494
C04281=1060.571,421.042,378.974,175.494,38.955,157.491
C04282=1060.562,420.796,379.019,175.486,38.945,157.488
C04283=1060.554,420.551,379.066,175.477,38.935,157.485
C04284=1060.545,420.305,379.111,175.470,38.925,157.483
C04285=1060.535,420.060,379.157,175.461,38.915,157.480
C04286=1060.527,419.814,379.203,175.453,38.905,157.477
C04287=1060.518,419.567,379.249,175.445,38.895,157.474
C04288=1060.509,419.322,379.294,175.437,38.886,157.472
C04289=1060.500,419.077,379.340,175.429,38.876,157.469
C04290=1060.491,418.831,379.386,175.421,38.866,157.466
C04291=1060.482,418.586,379.431,175.412,38.857,157.463
C04292=1060.473,418.340,379.476,175.405,38.847,157.461
C04293=1060.465,418.094,379.523,175.396,38.837,157.458
C04294=1060.456,417.848,379.568,175.389,38.827,157.455
C04295=1060.447,417.603,379.613,175.381,38.818,157.453
C04296=1060.439,417.357,379.658,175.373,38.808,157.450
C04297=1060.430,417.111,379.704,175.365,38.798,157.447
C04298=1060.421,416.865,379.749,175.358,38.789,157.445
C04299=1060.412,416.620,379.794,175.350,38.780,157.442
C04300=1060.403,416.374,379.840,175.342,38.770,157.439
C04301=1060.392,416.048,379.900,175.332,38.757,157.436
C04302=1060.380,415.722,379.960,175.322,38.745,157.433
C04303=1060.369,415.395,380.020,175.312,38.732,157.429
C04304=1060.358,415.070,380.079,175.302,38.720,157.426
C04305=1060.349,414.824,380.125,175.293,38.710,157.423
C04306=1060.341,414.578,380.169,175.286,38.701,157.420
C04307=1060.332,414.333,380.214,175.279,38.692,157.418
C04308=1060.323,414.086,380.259,175.271,38.683,157.415
C04309=1060.315,413.841,380.304,175.263,38.673,157.413
C04310=1060.306,413.595,380.348,175.256,38.664,157.410
C04311=1060.298,413.349,380.393,175.248,38.655,157.408
C04312=1060.289,413.103,380.438,175.241,38.646,157.405
C04313=1060.280,412.857,380.483,175.234,38.636,157.403
C04314=1060.272,412.611,380.527,175.226,38.628,157.400
C04315=1060.262,412.365,380.571,175.218,38.619,157.398
C04316=1060.254,412.120,380.616,175.211,38.610,157.396
C04317=1060.246,411.874,380.661,175.204,38.600,157.393
C04318=1060.237,411.628,380.705,175.197,38.591,157.391
C04319=1060.229,411.382,380.749,175.189,38.583,157.388
C04320=1060.220,411.136,380.794,175.182,38.574,157.386
C04321=1060.212,410.890,380.838,175.175,38.565,157.383
C04322=1060.203,410.645,380.882,175.167,38.556,157.381
C04323=1060.194,410.398,380.927,175.160,38.547,157.378
C04324=1060.186,410.153,380.971,175.153,38.538,157.376
C04325=1060.177,409.907,381.015,175.145,38.530,157.374
C04326=1060.169,409.660,381.059,175.138,38.521,157.371
C04327=1060.161,409.414,381.103,175.131,38.512,157.369
C04328=1060.153,409.169,381.147,175.124,38.503,157.367
C04329=1060.144,408.923,381.191,175.117,38.494,157.364
C04330=1060.136,408.676,381.235,175.110,38.486,157.362
C04331=1060.128,408.430,381.279,175.103,38.477,157.360
C04332=1060.119,408.185,381.323,175.096,38.468,157.357
C04333=1060.111,407.939,381.367,175.089,38.459,157.355
C04334=1060.103,407.693,381.411,175.082,38.451,157.353
C04335=1060.095,407.447,381.454,175.075,38.442,157.350
C04336=1060.087,407.201,381.498,175.068,38.434,157.348
C04337=1060.077,406.954,381.542,175.061,38.425,157.346
C04338=1060.069,406.708,381.586,175.054,38.417,157.343
C04339=1060.062,406.462,381.630,175.047,38.408,157.341
C04340=1060.053,406.217,381.674,175.041,38.400,157.339
C04341=1060.045,405.970,381.717,175.033,38.391,157.336
C04342=1060.037,405.724,381.761,175.027,38.382,157.334
C04343=1060.028,405.479,381.805,175.020,38.374,157.332
C04344=1060.021,405.232,381.848,175.013,38.366,157.330
C04345=1060.012,404.986,381.891,175.006,38.358,157.328
C04346=1060.004,404.740,381.934,175.000,38.349,157.325
C04347=1059.996,404.494,381.978,174.993,38.341,157.323
C04348=1059.987,404.248,382.021,174.986,38.333,157.321
C04349=1059.980,404.003,382.065,174.980,38.324,157.319
C04350=1059.971,403.757,382.108,174.973,38.316,157.317
C04351=1059.964,403.510,382.151,174.966,38.308,157.314
C04352=1059.955,403.264,382.195,174.959,38.300,157.312
C04353=1059.947,403.017,382.237,174.953,38.291,157.310
C04354=1059.939,402.771,382.280,174.947,38.283,157.308
C04355=1059.931,402.525,382.323,174.940,38.275,157.306
C04356=1059.922,402.279,382.366,174.933,38.267,157.303
C04357=1059.912,401.958,382.423,174.925,38.256,157.301
C04358=1059.902,401.638,382.479,174.916,38.246,157.298
C04359=1059.891,401.317,382.534,174.907,38.236,157.295
C04360=1059.880,400.996,382.590,174.899,38.225,157.292
C04361=1059.872,400.751,382.633,174.892,38.217,157.290
C04362=1059.864,400.504,382.675,174.886,38.209,157.288
C04363=1059.856,400.258,382.718,174.880,38.201,157.286
C04364=1059.848,400.012,382.760,174.873,38.193,157.284
C04365=1059.840,399.766,382.804,174.867,38.185,157.282
C04366=1059.832,399.519,382.846,174.860,38.177,157.280
C04367=1059.824,399.273,382.889,174.854,38.169,157.278
C04368=1059.816,399.027,382.931,174.847,38.162,157.276
C04369=1059.808,398.781,382.974,174.841,38.154,157.274
C04370=1059.800,398.535,383.016,174.835,38.146,157.272
C04371=1059.793,398.288,383.059,174.828,38.138,157.270
C04372=1059.784,398.042,383.102,174.822,38.131,157.268
C04373=1059.776,397.796,383.144,174.816,38.123,157.266
C04374=1059.768,397.550,383.186,174.809,38.115,157.264
C04375=1059.760,397.304,383.229,174.803,38.107,157.261
C04376=1059.752,397.057,383.271,174.797,38.100,157.260
C04377=1059.745,396.812,383.313,174.791,38.092,157.258
C04378=1059.736,396.565,383.355,174.785,38.085,157.256
C04379=1059.729,396.319,383.397,174.778,38.077,157.254
C04380=1059.721,396.072,383.440,174.772,38.069,157.252
C04381=1059.713,395.826,383.481,174.766,38.062,157.250
C04382=1059.705,395.580,383.524,174.760,38.054,157.248
C04383=1059.696,395.334,383.565,174.754,38.047,157.246
C04384=1059.689,395.088,383.607,174.747,38.039,157.244
C04385=1059.681,394.841,383.649,174.742,38.032,157.242
C04386=1059.673,394.595,383.691,174.735,38.024,157.240
C04387=1059.665,394.349,383.733,174.730,38.017,157.238
C04388=1059.657,394.103,383.776,174.723,38.009,157.236
C04389=1059.650,393.856,383.817,174.717,38.002,157.234
C04390=1059.642,393.610,383.859,174.711,37.994,157.232
C04391=1059.634,393.363,383.901,174.705,37.987,157.230
C04392=1059.626,393.118,383.942,174.699,37.979,157.228
C04393=1059.619,392.871,383.984,174.693,37.972,157.226
C04394=1059.611,392.625,384.026,174.687,37.965,157.225
C04395=1059.603,392.378,384.068,174.681,37.958,157.223
C04396=1059.595,392.132,384.109,174.675,37.950,157.221
C04397=1059.587,391.886,384.151,174.669,37.943,157.219
C04398=1059.580,391.640,384.192,174.663,37.936,157.217
C04399=1059.572,391.393,384.234,174.657,37.928,157.215
C04400=1059.564,391.147,384.275,174.651,37.921,157.213
C04401=1059.556,390.901,384.317,174.646,37.914,157.211
C04402=1059.549,390.654,384.358,174.639,37.907,157.210
C04403=1059.540,390.408,384.399,174.634,37.900,157.208
C04404=1059.533,390.162,384.440,174.627,37.893,157.206
C04405=1059.526,389.915,384.482,174.622,37.885,157.204
C04406=1059.517,389.668,384.523,174.616,37.878,157.202
C04407=1059.510,389.422,384.565,174.610,37.871,157.200
C04408=1059.502,389.176,384.605,174.604,37.864,157.199
C04409=1059.494,388.929,384.646,174.598,37.857,157.197
C04410=1059.486,388.683,384.687,174.593,37.850,157.195
C04411=1059.479,388.437,384.728,174.587,37.843,157.193
C04412=1059.471,388.190,384.769,174.581,37.836,157.191
C04413=1059.461,387.886,384.820,174.574,37.827,157.189
C04414=1059.452,387.583,384.871,174.566,37.819,157.187
C04415=1059.442,387.280,384.920,174.560,37.810,157.185
C04416=1059.432,386.977,384.971,174.553,37.802,157.183
C04417=1059.425,386.730,385.012,174.547,37.795,157.181
C04418=1059.417,386.483,385.052,174.541,37.788,157.179
C04419=1059.409,386.237,385.093,174.536,37.781,157.177
C04420=1059.402,385.990,385.134,174.530,37.774,157.176
C04421=1059.394,385.744,385.175,174.524,37.767,157.174
C04422=1059.387,385.497,385.216,174.519,37.760,157.172
C04423=1059.379,385.251,385.257,174.514,37.754,157.171
C04424=1059.372,385.004,385.297,174.507,37.747,157.169
C04425=1059.362,384.716,385.344,174.501,37.739,157.167
C04426=1059.353,384.426,385.392,174.494,37.731,157.165
C04427=1059.344,384.138,385.440,174.488,37.723,157.163
C04428=1059.336,383.849,385.487,174.481,37.715,157.161
C04429=1059.329,383.602,385.528,174.476,37.708,157.159
C04430=1059.321,383.356,385.569,174.471,37.702,157.157
C04431=1059.313,383.109,385.609,174.466,37.695,157.156
C04432=1059.306,382.863,385.650,174.459,37.688,157.154
C04433=1059.299,382.616,385.689,174.454,37.682,157.152
C04434=1059.291,382.370,385.731,174.449,37.675,157.151
C04435=1059.284,382.123,385.771,174.443,37.669,157.149
C04436=1059.276,381.877,385.811,174.438,37.662,157.147
C04437=1059.269,381.630,385.851,174.432,37.655,157.146
C04438=1059.261,381.383,385.891,174.427,37.649,157.144
C04439=1059.254,381.138,385.932,174.421,37.642,157.142
C04440=1059.247,380.890,385.972,174.416,37.636,157.141
C04441=1059.239,380.643,386.012,174.411,37.629,157.139
C04442=1059.232,380.397,386.052,174.406,37.623,157.137
C04443=1059.224,380.151,386.092,174.400,37.616,157.136
C04444=1059.216,379.904,386.132,174.394,37.609,157.134
C04445=1059.209,379.657,386.172,174.389,37.603,157.133
C04446=1059.202,379.411,386.212,174.384,37.596,157.131
C04447=1059.194,379.164,386.251,174.379,37.590,157.129
C04448=1059.186,378.917,386.291,174.374,37.584,157.128
C04449=1059.179,378.671,386.331,174.368,37.577,157.126
C04450=1059.171,378.424,386.371,174.362,37.571,157.125
C04451=1059.164,378.177,386.411,174.357,37.565,157.123
C04452=1059.156,377.931,386.450,174.352,37.558,157.121
C04453=1059.150,377.684,386.491,174.347,37.552,157.120
C04454=1059.142,377.438,386.530,174.341,37.546,157.118
C04455=1059.135,377.191,386.570,174.336,37.539,157.117
C04456=1059.128,376.944,386.610,174.331,37.533,157.115
C04457=1059.120,376.698,386.650,174.326,37.527,157.114
C04458=1059.112,376.450,386.689,174.321,37.521,157.112
C04459=1059.105,376.204,386.729,174.316,37.514,157.110
C04460=1059.098,375.957,386.768,174.311,37.508,157.109
C04461=1059.090,375.711,386.808,174.305,37.502,157.107
C04462=1059.082,375.463,386.847,174.300,37.495,157.106
C04463=1059.075,375.217,386.886,174.295,37.489,157.104
C04464=1059.068,374.971,386.926,174.290,37.483,157.103
C04465=1059.061,374.733,386.964,174.285,37.477,157.101
C04466=1059.054,374.494,387.003,174.280,37.471,157.100
C04467=1059.047,374.255,387.040,174.275,37.465,157.098
C04468=1059.040,374.017,387.078,174.270,37.459,157.097
C04469=1059.033,373.779,387.116,174.265,37.453,157.095
C04470=1059.026,373.541,387.154,174.260,37.447,157.094
C04471=1059.019,373.303,387.192,174.256,37.441,157.092
C04472=1059.012,373.065,387.231,174.251,37.436,157.091
C04473=1059.005,372.817,387.270,174.245,37.429,157.089
C04474=1058.998,372.570,387.309,174.240,37.423,157.088
C04475=1058.991,372.324,387.348,174.235,37.417,157.086
C04476=1058.983,372.077,387.387,174.230,37.411,157.085
C04477=1058.976,371.831,387.426,174.225,37.405,157.083
C04478=1058.969,371.584,387.465,174.220,37.399,157.082
C04479=1058.961,371.337,387.504,174.215,37.393,157.081
C04480=1058.954,371.090,387.543,174.210,37.388,157.079
C04481=1058.947,370.844,387.582,174.205,37.381,157.078
C04482=1058.939,370.596,387.621,174.200,37.375,157.076
C04483=1058.932,370.350,387.660,174.195,37.369,157.075
C04484=1058.925,370.103,387.698,174.190,37.363,157.073
C04485=1058.917,369.856,387.737,174.185,37.358,157.072
C04486=1058.910,369.609,387.776,174.180,37.352,157.070
C04487=1058.903,369.362,387.814,174.176,37.346,157.069
C04488=1058.896,369.115,387.853,174.171,37.340,157.068
C04489=1058.888,368.868,387.892,174.166,37.334,157.066
C04490=1058.881,368.621,387.930,174.161,37.328,157.065
C04491=1058.874,368.375,387.969,174.156,37.323,157.063
C04492=1058.867,368.128,388.008,174.151,37.317,157.062
C04493=1058.860,367.881,388.046,174.146,37.311,157.060
C04494=1058.852,367.634,388.086,174.141,37.305,157.059
C04495=1058.845,367.387,388.124,174.137,37.299,157.058
C04496=1058.838,367.140,388.163,174.132,37.293,157.056
C04497=1058.830,366.894,388.201,174.127,37.287,157.055
C04498=1058.823,366.647,388.240,174.122,37.282,157.053
C04499=1058.817,366.400,388.278,174.117,37.276,157.052
C04500=1058.809,366.153,388.316,174.112,37.270,157.051
C04501=1058.803,365.906,388.355,174.108,37.265,157.049
C04502=1058.795,365.660,388.393,174.103,37.259,157.048
C04503=1058.788,365.412,388.432,174.098,37.253,157.046
C04504=1058.781,365.165,388.470,174.093,37.248,157.045
C04505=1058.774,364.918,388.509,174.088,37.242,157.044
C04506=1058.767,364.671,388.547,174.084,37.236,157.042
C04507=1058.759,364.424,388.585,174.079,37.231,157.041
C04508=1058.753,364.177,388.624,174.074,37.224,157.039
C04509=1058.745,363.930,388.661,174.069,37.219,157.038
C04510=1058.739,363.684,388.700,174.064,37.213,157.037
C04511=1058.731,363.436,388.738,174.060,37.208,157.035
C04512=1058.724,363.190,388.776,174.055,37.202,157.034
C04513=1058.717,362.942,388.814,174.050,37.197,157.033
C04514=1058.710,362.696,388.852,174.045,37.191,157.031
C04515=1058.703,362.449,388.890,174.041,37.186,157.030
C04516=1058.696,362.201,388.928,174.036,37.180,157.029
C04517=1058.688,361.955,388.966,174.032,37.175,157.027
C04518=1058.681,361.708,389.004,174.027,37.169,157.026
C04519=1058.675,361.460,389.042,174.023,37.164,157.025
C04520=1058.667,361.214,389.080,174.018,37.158,157.023
C04521=1058.660,360.967,389.118,174.013,37.152,157.022
C04522=1058.653,360.719,389.155,174.008,37.147,157.021
C04523=1058.647,360.473,389.193,174.004,37.141,157.019
C04524=1058.639,360.226,389.231,173.999,37.136,157.018
C04525=1058.632,359.971,389.270,173.994,37.130,157.017
C04526=1058.625,359.718,389.309,173.989,37.125,157.015
C04527=1058.617,359.465,389.347,173.985,37.119,157.014
C04528=1058.610,359.210,389.386,173.981,37.114,157.013
C04529=1058.603,358.963,389.423,173.976,37.108,157.011
C04530=1058.596,358.716,389.461,173.971,37.103,157.010
C04531=1058.589,358.469,389.499,173.967,37.098,157.009
C04532=1058.582,358.222,389.536,173.962,37.092,157.008
C04533=1058.575,357.974,389.574,173.957,37.086,157.006
C04534=1058.568,357.728,389.611,173.953,37.081,157.005
C04535=1058.561,357.481,389.648,173.948,37.076,157.004
C04536=1058.554,357.234,389.686,173.944,37.071,157.003
C04537=1058.546,356.987,389.724,173.940,37.065,157.001
C04538=1058.540,356.739,389.762,173.935,37.060,157.000
C04539=1058.533,356.493,389.799,173.930,37.055,156.999
C04540=1058.526,356.246,389.836,173.926,37.050,156.997
C04541=1058.519,355.998,389.873,173.921,37.044,156.996
C04542=1058.512,355.751,389.911,173.918,37.039,156.995
C04543=1058.505,355.504,389.948,173.913,37.034,156.994
C04544=1058.498,355.257,389.985,173.908,37.029,156.992
C04545=1058.491,355.009,390.022,173.904,37.023,156.991
C04546=1058.484,354.762,390.060,173.899,37.018,156.990
C04547=1058.477,354.516,390.097,173.895,37.013,156.989
C04548=1058.470,354.268,390.134,173.890,37.007,156.987
C04549=1058.463,354.021,390.171,173.886,37.002,156.986
C04550=1058.456,353.774,390.208,173.882,36.997,156.985
C04551=1058.449,353.527,390.245,173.877,36.992,156.984
C04552=1058.442,353.280,390.283,173.873,36.987,156.983
C04553=1058.436,353.033,390.319,173.868,36.982,156.981
C04554=1058.428,352.785,390.357,173.864,36.976,156.980
C04555=1058.422,352.538,390.393,173.860,36.971,156.979
C04556=1058.415,352.291,390.431,173.855,36.966,156.978
C04557=1058.407,352.044,390.467,173.851,36.961,156.976
C04558=1058.400,351.797,390.504,173.846,36.956,156.975
C04559=1058.394,351.550,390.541,173.843,36.950,156.974
C04560=1058.387,351.303,390.578,173.838,36.945,156.973
C04561=1058.380,351.055,390.615,173.834,36.940,156.972
C04562=1058.373,350.808,390.652,173.829,36.935,156.970
C04563=1058.367,350.561,390.688,173.825,36.930,156.969
C04564=1058.359,350.314,390.725,173.821,36.925,156.968
C04565=1058.352,350.067,390.761,173.817,36.920,156.967
C04566=1058.345,349.819,390.798,173.812,36.915,156.966
C04567=1058.339,349.572,390.835,173.808,36.910,156.964
C04568=1058.331,349.325,390.872,173.804,36.905,156.963
C04569=1058.325,349.078,390.908,173.800,36.900,156.962
C04570=1058.318,348.830,390.945,173.795,36.895,156.961
C04571=1058.310,348.583,390.981,173.791,36.890,156.960
C04572=1058.304,348.336,391.018,173.786,36.885,156.959
C04573=1058.298,348.089,391.054,173.783,36.880,156.957
C04574=1058.290,347.842,391.092,173.778,36.875,156.956
C04575=1058.283,347.595,391.127,173.774,36.870,156.955
C04576=1058.276,347.347,391.164,173.769,36.865,156.954
C04577=1058.270,347.100,391.201,173.766,36.860,156.953
C04578=1058.262,346.853,391.237,173.761,36.855,156.952
C04579=1058.256,346.606,391.273,173.757,36.850,156.950
C04580=1058.249,346.358,391.310,173.753,36.846,156.949
C04581=1058.242,346.109,391.346,173.749,36.841,156.948
C04582=1058.235,345.860,391.382,173.744,36.836,156.947
C04583=1058.229,345.610,391.419,173.740,36.830,156.946
C04584=1058.222,345.361,391.455,173.735,36.825,156.945
C04585=1058.215,345.114,391.492,173.732,36.821,156.944
C04586=1058.208,344.867,391.528,173.728,36.816,156.942
C04587=1058.201,344.620,391.565,173.723,36.811,156.941
C04588=1058.194,344.373,391.600,173.720,36.806,156.940
C04589=1058.188,344.124,391.637,173.715,36.801,156.939
C04590=1058.181,343.877,391.673,173.711,36.796,156.938
C04591=1058.174,343.631,391.709,173.707,36.792,156.937
C04592=1058.167,343.383,391.746,173.703,36.787,156.936
C04593=1058.161,343.136,391.781,173.699,36.782,156.935
C04594=1058.154,342.888,391.817,173.694,36.777,156.933
C04595=1058.147,342.641,391.853,173.691,36.772,156.932
C04596=1058.140,342.393,391.889,173.687,36.767,156.931
C04597=1058.133,342.147,391.925,173.682,36.763,156.930
C04598=1058.126,341.899,391.960,173.678,36.758,156.929
C04599=1058.120,341.651,391.997,173.675,36.753,156.928
C04600=1058.113,341.404,392.032,173.670,36.748,156.927
C04601=1058.106,341.157,392.068,173.666,36.744,156.926
C04602=1058.099,340.909,392.104,173.662,36.739,156.925
C04603=1058.092,340.662,392.140,173.658,36.734,156.923
C04604=1058.085,340.415,392.175,173.654,36.730,156.922
C04605=1058.079,340.168,392.211,173.650,36.725,156.921
C04606=1058.072,339.920,392.247,173.646,36.720,156.920
C04607=1058.065,339.673,392.283,173.642,36.716,156.919
C04608=1058.059,339.425,392.319,173.638,36.710,156.918
C04609=1058.052,339.178,392.354,173.634,36.706,156.917
C04610=1058.045,338.931,392.390,173.630,36.701,156.916
C04611=1058.038,338.683,392.426,173.626,36.697,156.915
C04612=1058.031,338.435,392.461,173.622,36.692,156.914
C04613=1058.025,338.188,392.497,173.618,36.687,156.913
C04614=1058.018,337.941,392.532,173.615,36.683,156.912
C04615=1058.011,337.694,392.567,173.610,36.678,156.910
C04616=1058.005,337.446,392.603,173.606,36.673,156.909
C04617=1057.998,337.199,392.639,173.603,36.669,156.908
C04618=1057.992,336.952,392.674,173.598,36.664,156.907
C04619=1057.985,336.705,392.709,173.594,36.660,156.906
C04620=1057.977,336.456,392.745,173.591,36.654,156.905
C04621=1057.971,336.209,392.781,173.587,36.650,156.904
C04622=1057.965,335.961,392.816,173.582,36.645,156.903
C04623=1057.958,335.714,392.851,173.579,36.641,156.902
C04624=1057.951,335.467,392.886,173.575,36.636,156.901
C04625=1057.944,335.219,392.921,173.570,36.632,156.900
C04626=1057.938,334.972,392.956,173.567,36.627,156.899
C04627=1057.931,334.725,392.991,173.563,36.623,156.898
C04628=1057.924,334.477,393.026,173.560,36.618,156.897
C04629=1057.917,334.230,393.062,173.555,36.614,156.896
C04630=1057.911,333.983,393.097,173.551,36.609,156.895
C04631=1057.904,333.735,393.132,173.548,36.605,156.894
C04632=1057.898,333.488,393.168,173.544,36.600,156.893
C04633=1057.891,333.240,393.203,173.540,36.595,156.892
C04634=1057.884,332.993,393.238,173.536,36.591,156.891
C04635=1057.877,332.745,393.273,173.532,36.586,156.889
C04636=1057.871,332.498,393.308,173.528,36.582,156.888
C04637=1057.864,332.244,393.343,173.525,36.577,156.887
C04638=1057.856,331.991,393.379,173.520,36.573,156.886
C04639=1057.850,331.738,393.416,173.517,36.568,156.885
C04640=1057.843,331.483,393.451,173.513,36.564,156.884
C04641=1057.836,331.236,393.486,173.509,36.559,156.883
C04642=1057.830,330.989,393.521,173.505,36.555,156.882
C04643=1057.823,330.741,393.556,173.501,36.550,156.881
C04644=1057.817,330.494,393.590,173.497,36.545,156.880
C04645=1057.810,330.247,393.626,173.494,36.541,156.879
C04646=1057.804,329.999,393.660,173.490,36.537,156.878
C04647=1057.796,329.752,393.695,173.486,36.532,156.877
C04648=1057.790,329.504,393.729,173.482,36.528,156.876
C04649=1057.783,329.256,393.764,173.479,36.524,156.875
C04650=1057.776,329.009,393.798,173.475,36.519,156.874
C04651=1057.769,328.761,393.833,173.471,36.515,156.873
C04652=1057.763,328.513,393.867,173.468,36.511,156.872
C04653=1057.755,328.266,393.902,173.463,36.507,156.871
C04654=1057.749,328.018,393.936,173.460,36.502,156.870
C04655=1057.742,327.771,393.972,173.456,36.498,156.869
C04656=1057.735,327.523,394.005,173.452,36.494,156.868
C04657=1057.728,327.276,394.041,173.449,36.489,156.867
C04658=1057.722,327.029,394.075,173.445,36.485,156.866
C04659=1057.715,326.781,394.108,173.441,36.480,156.865
C04660=1057.708,326.534,394.144,173.437,36.476,156.865
C04661=1057.702,326.286,394.178,173.434,36.472,156.864
C04662=1057.694,326.038,394.212,173.430,36.468,156.863
C04663=1057.688,325.790,394.247,173.426,36.463,156.862
C04664=1057.682,325.543,394.281,173.423,36.459,156.861
C04665=1057.675,325.296,394.315,173.419,36.455,156.860
C04666=1057.668,325.048,394.349,173.416,36.451,156.859
C04667=1057.661,324.801,394.384,173.412,36.446,156.858
C04668=1057.655,324.553,394.418,173.408,36.442,156.857
C04669=1057.648,324.305,394.452,173.404,36.438,156.856
C04670=1057.641,324.058,394.486,173.401,36.434,156.855
C04671=1057.635,323.810,394.520,173.397,36.429,156.854
C04672=1057.628,323.563,394.555,173.393,36.425,156.853
C04673=1057.621,323.315,394.589,173.390,36.420,156.852
C04674=1057.615,323.067,394.624,173.386,36.416,156.851
C04675=1057.608,322.820,394.657,173.383,36.412,156.850
C04676=1057.602,322.572,394.691,173.379,36.408,156.849
C04677=1057.595,322.325,394.725,173.376,36.404,156.848
C04678=1057.589,322.077,394.759,173.372,36.399,156.847
C04679=1057.581,321.830,394.793,173.369,36.395,156.846
C04680=1057.575,321.582,394.828,173.365,36.391,156.845
C04681=1057.569,321.334,394.862,173.361,36.387,156.844
C04682=1057.562,321.087,394.895,173.358,36.383,156.844
C04683=1057.555,320.839,394.930,173.353,36.378,156.842
C04684=1057.549,320.592,394.963,173.350,36.374,156.842
C04685=1057.542,320.344,394.998,173.346,36.370,156.841
C04686=1057.536,320.097,395.031,173.343,36.365,156.840
C04687=1057.529,319.849,395.066,173.339,36.361,156.839
C04688=1057.522,319.601,395.099,173.336,36.357,156.838
C04689=1057.516,319.354,395.133,173.332,36.353,156.837
C04690=1057.509,319.106,395.167,173.329,36.349,156.836
C04691=1057.504,318.858,395.201,173.325,36.344,156.835
C04692=1057.496,318.611,395.234,173.321,36.340,156.834
C04693=1057.490,318.352,395.270,173.318,36.336,156.833
C04694=1057.483,318.093,395.305,173.314,36.332,156.832
C04695=1057.477,317.834,395.341,173.311,36.327,156.831
C04696=1057.470,317.575,395.377,173.307,36.323,156.830
C04697=1057.464,317.327,395.409,173.304,36.318,156.829
C04698=1057.457,317.079,395.444,173.300,36.314,156.828
C04699=1057.451,316.832,395.477,173.297,36.310,156.827
C04700=1057.445,316.585,395.511,173.293,36.306,156.827
C04701=1057.438,316.337,395.544,173.290,36.302,156.825
C04702=1057.432,316.090,395.578,173.286,36.298,156.825
C04703=1057.425,315.842,395.612,173.283,36.294,156.824
C04704=1057.418,315.594,395.645,173.279,36.290,156.823
C04705=1057.412,315.346,395.679,173.276,36.285,156.822
C04706=1057.406,315.099,395.712,173.272,36.281,156.821
C04707=1057.400,314.852,395.746,173.269,36.277,156.820
C04708=1057.393,314.604,395.780,173.266,36.273,156.819
C04709=1057.387,314.356,395.813,173.262,36.268,156.818
C04710=1057.380,314.109,395.847,173.259,36.264,156.817
C04711=1057.374,313.860,395.880,173.255,36.260,156.816
C04712=1057.368,313.613,395.914,173.252,36.256,156.815
C04713=1057.361,313.366,395.947,173.248,36.252,156.815
C04714=1057.355,313.117,395.980,173.245,36.248,156.814
C04715=1057.348,312.871,396.013,173.241,36.244,156.813
C04716=1057.341,312.622,396.046,173.238,36.240,156.812
C04717=1057.335,312.375,396.079,173.234,36.236,156.811
C04718=1057.328,312.127,396.113,173.231,36.232,156.810
C04719=1057.321,311.879,396.146,173.227,36.228,156.809
C04720=1057.314,311.631,396.179,173.224,36.224,156.808
C04721=1057.308,311.384,396.212,173.221,36.220,156.808
C04722=1057.301,311.137,396.245,173.217,36.216,156.807
C04723=1057.295,310.888,396.278,173.215,36.212,156.806
C04724=1057.288,310.641,396.311,173.211,36.208,156.805
C04725=1057.281,310.392,396.344,173.208,36.204,156.804
C04726=1057.275,310.145,396.377,173.204,36.200,156.803
C04727=1057.269,309.898,396.410,173.201,36.196,156.802
C04728=1057.262,309.649,396.443,173.197,36.192,156.801
C04729=1057.255,309.402,396.475,173.194,36.189,156.801
C04730=1057.248,309.155,396.508,173.190,36.185,156.800
C04731=1057.242,308.907,396.541,173.187,36.181,156.799
C04732=1057.235,308.659,396.574,173.183,36.177,156.798
C04733=1057.228,308.412,396.607,173.181,36.173,156.797
C04734=1057.222,308.164,396.640,173.177,36.168,156.796
C04735=1057.215,307.916,396.673,173.174,36.165,156.795
C04736=1057.209,307.668,396.706,173.170,36.161,156.794
C04737=1057.203,307.421,396.739,173.167,36.157,156.794
C04738=1057.196,307.173,396.771,173.163,36.153,156.793
C04739=1057.189,306.925,396.804,173.160,36.149,156.792
C04740=1057.183,306.677,396.837,173.157,36.145,156.791
C04741=1057.176,306.430,396.870,173.154,36.141,156.790
C04742=1057.170,306.182,396.902,173.151,36.137,156.789
C04743=1057.164,305.935,396.935,173.147,36.133,156.788
C04744=1057.157,305.687,396.968,173.144,36.129,156.788
C04745=1057.151,305.438,397.000,173.140,36.126,156.787
C04746=1057.144,305.191,397.032,173.137,36.122,156.786
C04747=1057.137,304.943,397.065,173.134,36.117,156.785
C04748=1057.131,304.696,397.098,173.131,36.113,156.784
C04749=1057.125,304.440,397.132,173.127,36.109,156.783
C04750=1057.118,304.186,397.165,173.124,36.105,156.782
C04751=1057.111,303.931,397.199,173.120,36.101,156.781
C04752=1057.105,303.677,397.232,173.117,36.097,156.781
C04753=1057.099,303.429,397.264,173.114,36.094,156.780
C04754=1057.093,303.181,397.297,173.111,36.090,156.779
C04755=1057.085,302.933,397.329,173.108,36.086,156.778
C04756=1057.079,302.686,397.362,173.104,36.082,156.777
C04757=1057.073,302.438,397.394,173.101,36.078,156.776
C04758=1057.066,302.190,397.427,173.098,36.074,156.776
C04759=1057.060,301.942,397.460,173.095,36.070,156.775
C04760=1057.054,301.694,397.492,173.091,36.066,156.774
C04761=1057.047,301.447,397.524,173.088,36.062,156.773
C04762=1057.041,301.199,397.557,173.084,36.058,156.772
C04763=1057.035,300.951,397.589,173.082,36.054,156.771
C04764=1057.028,300.703,397.621,173.079,36.050,156.770
C04765=1057.022,300.456,397.654,173.075,36.047,156.770
C04766=1057.015,300.208,397.685,173.072,36.043,156.769
C04767=1057.009,299.960,397.718,173.069,36.039,156.768
C04768=1057.003,299.712,397.750,173.066,36.035,156.767
C04769=1056.997,299.465,397.783,173.062,36.031,156.766
C04770=1056.990,299.217,397.814,173.060,36.027,156.765
C04771=1056.984,298.969,397.847,173.056,36.023,156.765
C04772=1056.978,298.721,397.879,173.053,36.019,156.764
C04773=1056.972,298.473,397.912,173.050,36.015,156.763
C04774=1056.966,298.225,397.944,173.047,36.011,156.762
C04775=1056.959,297.978,397.976,173.044,36.008,156.761
C04776=1056.953,297.730,398.008,173.040,36.004,156.760
C04777=1056.947,297.483,398.040,173.038,36.000,156.759
C04778=1056.941,297.234,398.073,173.034,35.996,156.759
C04779=1056.934,296.987,398.104,173.031,35.992,156.758
C04780=1056.928,296.739,398.137,173.028,35.988,156.757
C04781=1056.922,296.491,398.169,173.025,35.984,156.756
C04782=1056.915,296.243,398.200,173.022,35.980,156.755
C04783=1056.909,295.995,398.233,173.018,35.977,156.755
C04784=1056.902,295.747,398.264,173.016,35.973,156.754
C04785=1056.896,295.499,398.296,173.012,35.969,156.753
C04786=1056.889,295.251,398.328,173.009,35.965,156.752
C04787=1056.884,295.004,398.360,173.007,35.962,156.751
C04788=1056.877,294.756,398.392,173.003,35.958,156.750
C04789=1056.870,294.509,398.423,173.000,35.954,156.750
C04790=1056.864,294.260,398.455,172.997,35.950,156.749
C04791=1056.858,294.012,398.486,172.994,35.946,156.748
C04792=1056.852,293.764,398.519,172.990,35.942,156.747
C04793=1056.845,293.517,398.551,172.987,35.939,156.746
C04794=1056.838,293.269,398.582,172.985,35.935,156.746
C04795=1056.832,293.021,398.614,172.981,35.931,156.745
C04796=1056.825,292.773,398.646,172.978,35.927,156.744
C04797=1056.819,292.526,398.677,172.975,35.924,156.743
C04798=1056.813,292.277,398.709,172.972,35.920,156.742
C04799=1056.806,292.030,398.740,172.970,35.916,156.742
C04800=1056.800,291.782,398.772,172.966,35.913,156.741
C04801=1056.794,291.538,398.802,172.963,35.908,156.740
C04802=1056.788,291.294,398.833,172.960,35.905,156.739
C04803=1056.781,291.051,398.864,172.957,35.901,156.738
C04804=1056.775,290.807,398.896,172.955,35.897,156.738
C04805=1056.769,290.564,398.926,172.951,35.894,156.737
C04806=1056.762,290.321,398.957,172.948,35.890,156.736
C04807=1056.756,290.077,398.988,172.945,35.887,156.735
C04808=1056.750,289.834,399.019,172.942,35.883,156.734
C04809=1056.743,289.586,399.051,172.940,35.879,156.734
C04810=1056.737,289.338,399.082,172.936,35.876,156.733
C04811=1056.731,289.091,399.113,172.933,35.872,156.732
C04812=1056.724,288.842,399.144,172.930,35.868,156.731
C04813=1056.718,288.594,399.176,172.927,35.864,156.730
C04814=1056.711,288.346,399.207,172.925,35.860,156.730
C04815=1056.705,288.099,399.238,172.921,35.857,156.729
C04816=1056.699,287.851,399.270,172.918,35.853,156.728
C04817=1056.692,287.602,399.301,172.916,35.849,156.727
C04818=1056.685,287.354,399.332,172.912,35.846,156.727
C04819=1056.679,287.107,399.363,172.910,35.842,156.726
C04820=1056.673,286.859,399.394,172.906,35.838,156.725
C04821=1056.667,286.610,399.426,172.903,35.835,156.724
C04822=1056.660,286.363,399.457,172.901,35.831,156.723
C04823=1056.654,286.115,399.488,172.897,35.827,156.723
C04824=1056.648,285.867,399.519,172.895,35.824,156.722
C04825=1056.641,285.619,399.550,172.891,35.820,156.721
C04826=1056.635,285.370,399.581,172.888,35.816,156.720
C04827=1056.628,285.123,399.612,172.886,35.812,156.720
C04828=1056.622,284.875,399.643,172.882,35.809,156.719
C04829=1056.615,284.627,399.674,172.880,35.805,156.718
C04830=1056.609,284.379,399.705,172.876,35.801,156.717
C04831=1056.603,284.131,399.736,172.874,35.798,156.716
C04832=1056.596,283.883,399.767,172.871,35.794,156.716
C04833=1056.590,283.635,399.798,172.868,35.791,156.715
C04834=1056.584,283.387,399.829,172.865,35.787,156.714
C04835=1056.577,283.139,399.860,172.862,35.783,156.713
C04836=1056.571,282.891,399.890,172.859,35.779,156.713
C04837=1056.564,282.643,399.922,172.856,35.775,156.712
C04838=1056.559,282.395,399.952,172.853,35.772,156.711
C04839=1056.552,282.147,399.984,172.850,35.768,156.710
C04840=1056.546,281.899,400.014,172.848,35.765,156.709
C04841=1056.540,281.651,400.045,172.844,35.761,156.709
C04842=1056.533,281.403,400.076,172.842,35.757,156.708
C04843=1056.527,281.155,400.107,172.839,35.754,156.707
C04844=1056.520,280.907,400.138,172.836,35.750,156.706
C04845=1056.515,280.660,400.168,172.833,35.746,156.706
C04846=1056.508,280.411,400.199,172.830,35.742,156.705
C04847=1056.501,280.163,400.230,172.827,35.739,156.704
C04848=1056.496,279.915,400.261,172.825,35.735,156.703
C04849=1056.489,279.667,400.292,172.821,35.731,156.702
C04850=1056.483,279.419,400.322,172.819,35.728,156.702
C04851=1056.476,279.171,400.352,172.816,35.724,156.701
C04852=1056.470,278.924,400.383,172.813,35.721,156.700
C04853=1056.464,278.675,400.414,172.810,35.717,156.699
C04854=1056.457,278.427,400.445,172.808,35.713,156.699
C04855=1056.451,278.179,400.474,172.804,35.709,156.698
C04856=1056.444,277.931,400.505,172.802,35.706,156.697
C04857=1056.439,277.693,400.534,172.798,35.702,156.696
C04858=1056.432,277.455,400.563,172.796,35.699,156.696
C04859=1056.426,277.217,400.593,172.794,35.695,156.695
C04860=1056.420,276.979,400.622,172.790,35.692,156.694
C04861=1056.414,276.742,400.651,172.788,35.688,156.693
C04862=1056.408,276.503,400.680,172.786,35.685,156.693
C04863=1056.403,276.264,400.710,172.782,35.682,156.692
C04864=1056.396,276.027,400.740,172.780,35.678,156.691
C04865=1056.390,275.779,400.769,172.777,35.675,156.691
C04866=1056.383,275.531,400.800,172.774,35.670,156.690
C04867=1056.377,275.283,400.830,172.772,35.667,156.689
C04868=1056.370,275.035,400.861,172.769,35.663,156.688
C04869=1056.364,274.787,400.891,172.766,35.660,156.687
C04870=1056.359,274.539,400.921,172.763,35.656,156.687
C04871=1056.351,274.291,400.951,172.761,35.653,156.686
C04872=1056.346,274.043,400.982,172.757,35.649,156.685
C04873=1056.339,273.794,401.012,172.755,35.645,156.684
C04874=1056.333,273.546,401.041,172.753,35.642,156.684
C04875=1056.326,273.298,401.072,172.749,35.638,156.683
C04876=1056.321,273.050,401.103,172.747,35.634,156.682
C04877=1056.314,272.802,401.132,172.744,35.631,156.681
C04878=1056.308,272.554,401.163,172.741,35.627,156.681
C04879=1056.301,272.306,401.193,172.738,35.624,156.680
C04880=1056.295,272.057,401.223,172.736,35.620,156.679
C04881=1056.288,271.810,401.252,172.733,35.616,156.678
C04882=1056.282,271.561,401.283,172.730,35.613,156.678
C04883=1056.276,271.313,401.314,172.727,35.609,156.677
C04884=1056.270,271.065,401.343,172.724,35.605,156.676
C04885=1056.264,270.817,401.373,172.722,35.602,156.675
C04886=1056.257,270.569,401.403,172.719,35.598,156.675
C04887=1056.251,270.321,401.433,172.716,35.595,156.674
C04888=1056.244,270.073,401.463,172.714,35.591,156.673
C04889=1056.238,269.825,401.493,172.710,35.588,156.672
C04890=1056.231,269.577,401.523,172.708,35.584,156.672
C04891=1056.225,269.328,401.552,172.706,35.581,156.671
C04892=1056.219,269.081,401.583,172.702,35.577,156.670
C04893=1056.212,268.832,401.612,172.700,35.573,156.669
C04894=1056.207,268.584,401.642,172.698,35.569,156.669
C04895=1056.200,268.336,401.672,172.694,35.566,156.668
C04896=1056.194,268.087,401.702,172.692,35.562,156.667
C04897=1056.187,267.840,401.732,172.689,35.559,156.666
C04898=1056.181,267.592,401.761,172.686,35.555,156.666
C04899=1056.175,267.343,401.792,172.684,35.552,156.665
C04900=1056.168,267.095,401.821,172.681,35.548,156.664
C04901=1056.162,266.847,401.851,172.678,35.544,156.664
C04902=1056.156,266.599,401.880,172.676,35.541,156.663
C04903=1056.149,266.351,401.910,172.673,35.537,156.662
C04904=1056.143,266.103,401.939,172.670,35.534,156.661
C04905=1056.137,265.855,401.970,172.668,35.530,156.661
C04906=1056.130,265.606,401.999,172.665,35.527,156.660
C04907=1056.124,265.358,402.028,172.662,35.523,156.659
C04908=1056.118,265.110,402.058,172.660,35.520,156.658
C04909=1056.112,264.862,402.088,172.657,35.516,156.658
C04910=1056.105,264.614,402.118,172.654,35.512,156.657
C04911=1056.099,264.365,402.147,172.652,35.509,156.656
C04912=1056.093,264.117,402.176,172.649,35.505,156.655
C04913=1056.087,263.881,402.205,172.646,35.502,156.655
C04914=1056.081,263.645,402.233,172.644,35.498,156.654
C04915=1056.074,263.409,402.261,172.642,35.495,156.653
C04916=1056.069,263.174,402.289,172.640,35.492,156.653
C04917=1056.063,262.937,402.316,172.636,35.488,156.652
C04918=1056.057,262.701,402.345,172.634,35.485,156.651
C04919=1056.051,262.465,402.373,172.632,35.482,156.651
C04920=1056.045,262.229,402.401,172.629,35.478,156.650
C04921=1056.039,261.981,402.430,172.626,35.474,156.649
C04922=1056.032,261.732,402.459,172.624,35.471,156.648
C04923=1056.025,261.484,402.488,172.621,35.467,156.648
C04924=1056.019,261.236,402.518,172.619,35.464,156.647
C04925=1056.013,260.988,402.547,172.616,35.461,156.646
C04926=1056.005,260.739,402.575,172.613,35.457,156.646
C04927=1055.999,260.492,402.605,172.611,35.454,156.645
C04928=1055.993,260.244,402.634,172.608,35.450,156.644
C04929=1055.986,259.996,402.663,172.606,35.446,156.643
C04930=1055.979,259.747,402.693,172.603,35.443,156.643
C04931=1055.973,259.499,402.722,172.601,35.439,156.642
C04932=1055.967,259.251,402.751,172.598,35.436,156.641
C04933=1055.961,259.002,402.780,172.595,35.432,156.640
C04934=1055.954,258.754,402.809,172.593,35.429,156.640
C04935=1055.948,258.506,402.838,172.590,35.425,156.639
C04936=1055.941,258.257,402.867,172.587,35.422,156.638
C04937=1055.935,258.009,402.896,172.585,35.419,156.638
C04938=1055.929,257.761,402.925,172.583,35.415,156.637
C04939=1055.923,257.513,402.954,172.579,35.411,156.636
C04940=1055.916,257.265,402.983,172.577,35.408,156.635
C04941=1055.910,257.017,403.012,172.575,35.404,156.635
C04942=1055.904,256.769,403.041,172.573,35.401,156.634
C04943=1055.897,256.520,403.071,172.569,35.397,156.633
C04944=1055.890,256.271,403.099,172.567,35.394,156.633
C04945=1055.884,256.023,403.128,172.565,35.390,156.632
C04946=1055.878,255.775,403.157,172.562,35.386,156.631
C04947=1055.872,255.527,403.186,172.559,35.383,156.630
C04948=1055.865,255.279,403.215,172.557,35.379,156.630
C04949=1055.859,255.031,403.244,172.554,35.376,156.629
C04950=1055.853,254.782,403.273,172.552,35.372,156.628
C04951=1055.847,254.534,403.301,172.550,35.368,156.627
C04952=1055.841,254.286,403.330,172.546,35.365,156.627
C04953=1055.834,254.037,403.359,172.544,35.361,156.626
C04954=1055.827,253.790,403.388,172.542,35.358,156.625
C04955=1055.821,253.541,403.416,172.540,35.354,156.624
C04956=1055.815,253.293,403.445,172.537,35.351,156.624
C04957=1055.809,253.045,403.474,172.534,35.347,156.623
C04958=1055.803,252.796,403.503,172.532,35.343,156.622
C04959=1055.797,252.548,403.531,172.529,35.340,156.622
C04960=1055.791,252.300,403.560,172.527,35.336,156.621
C04961=1055.784,252.051,403.590,172.525,35.333,156.620
C04962=1055.778,251.803,403.618,172.521,35.329,156.619
C04963=1055.771,251.555,403.646,172.519,35.326,156.619
C04964=1055.765,251.307,403.675,172.517,35.322,156.618
C04965=1055.759,251.058,403.704,172.515,35.318,156.617
C04966=1055.753,250.810,403.733,172.512,35.315,156.616
C04967=1055.747,250.562,403.762,172.510,35.311,156.616
C04968=1055.741,250.313,403.790,172.508,35.308,156.615
C04969=1055.734,250.077,403.817,172.504,35.305,156.614
C04970=1055.728,249.839,403.845,172.502,35.301,156.614
C04971=1055.723,249.602,403.872,172.500,35.297,156.613
C04972=1055.717,249.365,403.900,172.497,35.294,156.612
C04973=1055.711,249.129,403.927,172.495,35.291,156.612
C04974=1055.705,248.891,403.954,172.493,35.287,156.611
C04975=1055.699,248.654,403.982,172.491,35.284,156.610
C04976=1055.693,248.417,404.008,172.488,35.280,156.609
C04977=1055.687,248.169,404.037,172.486,35.277,156.609
C04978=1055.681,247.920,404.065,172.484,35.273,156.608
C04979=1055.675,247.673,404.094,172.481,35.269,156.607
C04980=1055.669,247.424,404.122,172.479,35.266,156.607
C04981=1055.662,247.176,404.151,172.477,35.262,156.606
C04982=1055.656,246.927,404.179,172.474,35.259,156.605
C04983=1055.650,246.679,404.208,172.471,35.255,156.604
C04984=1055.644,246.431,404.237,172.469,35.251,156.604
C04985=1055.639,246.182,404.265,172.467,35.248,156.603
C04986=1055.632,245.935,404.293,172.464,35.244,156.602
C04987=1055.626,245.686,404.321,172.462,35.241,156.601
C04988=1055.620,245.437,404.350,172.460,35.237,156.601
C04989=1055.613,245.189,404.378,172.458,35.234,156.600
C04990=1055.607,244.941,404.406,172.455,35.230,156.599
C04991=1055.600,244.692,404.434,172.452,35.226,156.599
C04992=1055.594,244.444,404.463,172.450,35.223,156.598
C04993=1055.589,244.196,404.491,172.447,35.219,156.597
C04994=1055.582,243.948,404.519,172.445,35.216,156.596
C04995=1055.576,243.699,404.547,172.443,35.212,156.596
C04996=1055.569,243.451,404.576,172.441,35.208,156.595
C04997=1055.563,243.202,404.604,172.438,35.205,156.594
C04998=1055.556,242.954,404.632,172.436,35.201,156.593
C04999=1055.551,242.706,404.660,172.434,35.198,156.593
C05000=1055.545,242.457,404.688,172.431,35.194,156.592
C05001=1055.538,242.209,404.716,172.429,35.190,156.591
C05002=1055.532,241.960,404.745,172.427,35.187,156.591
C05003=1055.525,241.712,404.772,172.425,35.183,156.590
C05004=1055.519,241.464,404.800,172.421,35.180,156.589
C05005=1055.513,241.215,404.828,172.419,35.176,156.588
C05006=1055.507,240.967,404.856,172.417,35.172,156.588
C05007=1055.500,240.719,404.884,172.414,35.169,156.587
C05008=1055.494,240.470,404.912,172.412,35.165,156.586
C05009=1055.488,240.222,404.939,172.410,35.162,156.586
C05010=1055.482,239.973,404.968,172.408,35.159,156.585
C05011=1055.475,239.725,404.995,172.405,35.155,156.584
C05012=1055.469,239.476,405.023,172.403,35.152,156.583
C05013=1055.463,239.228,405.051,172.401,35.148,156.583
C05014=1055.457,238.980,405.079,172.399,35.144,156.582
C05015=1055.450,238.732,405.107,172.396,35.141,156.581
C05016=1055.443,238.483,405.134,172.394,35.137,156.581
C05017=1055.437,238.234,405.163,172.392,35.134,156.580
C05018=1055.431,237.987,405.190,172.389,35.130,156.579
C05019=1055.425,237.738,405.218,172.387,35.126,156.578
C05020=1055.419,237.489,405.246,172.385,35.123,156.578
C05021=1055.412,237.241,405.274,172.383,35.119,156.577
C05022=1055.406,236.993,405.301,172.380,35.116,156.576
C05023=1055.399,236.745,405.329,172.378,35.112,156.576
C05024=1055.394,236.495,405.356,172.376,35.108,156.575
C05025=1055.387,236.256,405.383,172.374,35.105,156.574
C05026=1055.381,236.016,405.410,172.371,35.102,156.573
C05027=1055.375,235.777,405.437,172.369,35.098,156.573
C05028=1055.369,235.536,405.463,172.367,35.095,156.572
C05029=1055.363,235.296,405.490,172.365,35.091,156.571
C05030=1055.357,235.056,405.517,172.362,35.088,156.571
C05031=1055.351,234.816,405.543,172.360,35.084,156.570
C05032=1055.345,234.576,405.570,172.358,35.081,156.569
C05033=1055.339,234.328,405.597,172.356,35.077,156.569
C05034=1055.333,234.079,405.626,172.353,35.074,156.568
C05035=1055.326,233.831,405.653,172.351,35.070,156.567
C05036=1055.320,233.582,405.680,172.349,35.066,156.566
C05037=1055.314,233.334,405.708,172.346,35.063,156.566
C05038=1055.308,233.086,405.736,172.344,35.059,156.565
C05039=1055.302,232.837,405.763,172.342,35.055,156.564
C05040=1055.295,232.588,405.790,172.340,35.052,156.564
C05041=1055.289,232.340,405.818,172.337,35.048,156.563
C05042=1055.283,232.091,405.845,172.335,35.045,156.562
C05043=1055.276,231.843,405.872,172.333,35.041,156.561
C05044=1055.270,231.595,405.900,172.331,35.037,156.561
C05045=1055.264,231.346,405.927,172.328,35.034,156.560
C05046=1055.258,231.098,405.955,172.326,35.030,156.559
C05047=1055.252,230.849,405.982,172.324,35.027,156.558
C05048=1055.245,230.601,406.010,172.323,35.023,156.558
C05049=1055.239,230.353,406.037,172.320,35.019,156.557
C05050=1055.233,230.104,406.064,172.318,35.016,156.556
C05051=1055.227,229.856,406.091,172.316,35.012,156.556
C05052=1055.220,229.607,406.118,172.314,35.009,156.555
C05053=1055.214,229.359,406.146,172.311,35.005,156.554
C05054=1055.208,229.110,406.173,172.309,35.001,156.553
C05055=1055.201,228.862,406.200,172.307,34.998,156.553
C05056=1055.195,228.613,406.227,172.304,34.994,156.552
C05057=1055.189,228.365,406.255,172.302,34.991,156.551
C05058=1055.183,228.117,406.281,172.300,34.987,156.551
C05059=1055.176,227.868,406.308,172.298,34.983,156.550
C05060=1055.169,227.619,406.336,172.295,34.980,156.549
C05061=1055.163,227.371,406.362,172.293,34.976,156.548
C05062=1055.157,227.123,406.390,172.291,34.973,156.548
C05063=1055.151,226.874,406.417,172.289,34.969,156.547
C05064=1055.145,226.625,406.444,172.287,34.965,156.546
C05065=1055.138,226.377,406.471,172.285,34.962,156.546
C05066=1055.132,226.128,406.498,172.283,34.959,156.545
C05067=1055.126,225.880,406.524,172.281,34.955,156.544
C05068=1055.119,225.632,406.552,172.278,34.951,156.544
C05069=1055.113,225.384,406.578,172.276,34.948,156.543
C05070=1055.107,225.134,406.605,172.274,34.944,156.542
C05071=1055.101,224.887,406.633,172.272,34.941,156.541
C05072=1055.094,224.638,406.660,172.269,34.936,156.541
C05073=1055.089,224.389,406.686,172.267,34.933,156.540
C05074=1055.081,224.141,406.713,172.265,34.929,156.539
C05075=1055.075,223.893,406.740,172.264,34.926,156.538
C05076=1055.069,223.644,406.767,172.261,34.922,156.538
C05077=1055.063,223.395,406.794,172.259,34.918,156.537
C05078=1055.057,223.146,406.821,172.257,34.915,156.536
C05079=1055.051,222.899,406.848,172.255,34.911,156.536
C05080=1055.044,222.650,406.875,172.252,34.907,156.535
C05081=1055.038,222.406,406.900,172.250,34.904,156.534
C05082=1055.032,222.162,406.927,172.249,34.900,156.533
C05083=1055.026,221.919,406.954,172.247,34.897,156.533
C05084=1055.020,221.674,406.980,172.244,34.893,156.532
C05085=1055.014,221.430,407.006,172.242,34.889,156.531
C05086=1055.007,221.187,407.033,172.240,34.886,156.531
C05087=1055.001,220.942,407.058,172.238,34.882,156.530
C05088=1054.995,220.699,407.085,172.236,34.879,156.529
C05089=1054.989,220.450,407.111,172.234,34.875,156.528
C05090=1054.983,220.201,407.138,172.232,34.871,156.528
C05091=1054.976,219.953,407.165,172.230,34.868,156.527
C05092=1054.970,219.705,407.191,172.228,34.865,156.526
C05093=1054.963,219.456,407.218,172.225,34.861,156.526
C05094=1054.958,219.208,407.244,172.224,34.857,156.525
C05095=1054.950,218.959,407.271,172.222,34.853,156.524
C05096=1054.945,218.711,407.297,172.220,34.850,156.523
C05097=1054.939,218.462,407.324,172.217,34.846,156.523
C05098=1054.932,218.214,407.350,172.215,34.842,156.522
C05099=1054.926,217.965,407.377,172.213,34.839,156.521
C05100=1054.919,217.716,407.403,172.212,34.835,156.521
C05101=1054.913,217.468,407.430,172.209,34.832,156.520
C05102=1054.907,217.220,407.456,172.207,34.828,156.519
C05103=1054.900,216.971,407.483,172.205,34.824,156.518
C05104=1054.894,216.723,407.510,172.203,34.821,156.518
C05105=1054.888,216.474,407.535,172.200,34.817,156.517
C05106=1054.882,216.225,407.562,172.199,34.813,156.516
C05107=1054.875,215.977,407.588,172.197,34.810,156.516
C05108=1054.870,215.728,407.615,172.195,34.806,156.515
C05109=1054.862,215.480,407.641,172.193,34.803,156.514
C05110=1054.857,215.231,407.668,172.190,34.799,156.513
C05111=1054.850,214.983,407.694,172.189,34.795,156.513
C05112=1054.844,214.734,407.720,172.187,34.791,156.512
C05113=1054.838,214.486,407.746,172.185,34.787,156.511
C05114=1054.832,214.237,407.773,172.182,34.784,156.510
C05115=1054.825,213.988,407.799,172.180,34.780,156.510
C05116=1054.819,213.739,407.825,172.179,34.777,156.509
C05117=1054.813,213.491,407.851,172.177,34.773,156.508
C05118=1054.807,213.243,407.878,172.174,34.769,156.508
C05119=1054.800,212.994,407.904,172.172,34.765,156.507
C05120=1054.794,212.745,407.930,172.171,34.762,156.506
C05121=1054.788,212.497,407.956,172.169,34.758,156.505
C05122=1054.782,212.249,407.983,172.166,34.754,156.505
C05123=1054.775,212.000,408.010,172.164,34.751,156.504
C05124=1054.769,211.751,408.035,172.163,34.747,156.503
C05125=1054.763,211.503,408.062,172.161,34.743,156.502
C05126=1054.756,211.255,408.088,172.159,34.740,156.502
C05127=1054.750,211.005,408.114,172.156,34.736,156.501
C05128=1054.744,210.757,408.140,172.154,34.732,156.500
C05129=1054.738,210.509,408.165,172.153,34.728,156.500
C05130=1054.732,210.260,408.192,172.151,34.725,156.499
C05131=1054.725,210.012,408.218,172.148,34.721,156.498
C05132=1054.719,209.763,408.244,172.146,34.717,156.497
C05133=1054.713,209.515,408.270,172.145,34.714,156.497
C05134=1054.707,209.266,408.296,172.143,34.710,156.496
C05135=1054.699,209.017,408.322,172.140,34.706,156.495
C05136=1054.694,208.768,408.348,172.138,34.702,156.494
C05137=1054.688,208.528,408.373,172.137,34.699,156.494
C05138=1054.682,208.286,408.398,172.135,34.695,156.493
C05139=1054.675,208.045,408.423,172.133,34.691,156.492
C05140=1054.669,207.804,408.448,172.131,34.688,156.492
C05141=1054.663,207.562,408.474,172.129,34.684,156.491
C05142=1054.657,207.321,408.498,172.127,34.681,156.490
C05143=1054.651,207.080,408.524,172.126,34.678,156.490
C05144=1054.644,206.838,408.549,172.124,34.674,156.489
C05145=1054.619,205.787,408.655,171.916,34.582,156.474
C05146=1054.614,205.539,408.679,171.914,34.579,156.474
C05147=1054.607,205.290,408.704,171.911,34.576,156.473
C05148=1054.602,205.041,408.729,171.908,34.573,156.473
C05149=1054.596,204.793,408.754,171.906,34.571,156.472
C05150=1054.590,204.544,408.779,171.904,34.567,156.472
C05151=1054.584,204.295,408.804,171.901,34.564,156.471
C05152=1054.577,204.047,408.828,171.899,34.562,156.471
C05153=1054.572,203.798,408.853,171.897,34.559,156.470
C05154=1054.565,203.549,408.878,171.895,34.556,156.470
C05155=1054.560,203.301,408.902,171.891,34.553,156.469
C05156=1054.554,203.052,408.928,171.889,34.550,156.468
C05157=1054.548,202.803,408.952,171.887,34.548,156.468
C05158=1054.542,202.555,408.977,171.884,34.544,156.467
C05159=1054.536,202.305,409.002,171.882,34.542,156.467
C05160=1054.530,202.057,409.027,171.880,34.539,156.466
C05161=1054.524,201.809,409.051,171.878,34.536,156.466
C05162=1054.518,201.559,409.075,171.874,34.533,156.465
C05163=1054.512,201.311,409.101,171.872,34.530,156.465
C05164=1054.506,201.062,409.124,171.870,34.528,156.464
C05165=1054.500,200.813,409.149,171.868,34.525,156.464
C05166=1054.493,200.565,409.174,171.865,34.522,156.463
C05167=1054.488,200.316,409.198,171.863,34.519,156.463
C05168=1054.482,200.067,409.223,171.861,34.516,156.462
C05169=1054.475,199.818,409.247,171.858,34.514,156.462
C05170=1054.470,199.570,409.272,171.855,34.511,156.461
C05171=1054.463,199.321,409.296,171.853,34.508,156.461
C05172=1054.457,199.072,409.321,171.851,34.506,156.460
C05173=1054.451,198.824,409.345,171.849,34.503,156.460
C05174=1054.445,198.575,409.369,171.846,34.500,156.459
C05175=1054.440,198.326,409.394,171.844,34.497,156.459
C05176=1054.433,198.077,409.418,171.842,34.495,156.458
C05177=1054.427,197.828,409.443,171.839,34.492,156.458
C05178=1054.421,197.580,409.467,171.836,34.489,156.457
C05179=1054.415,197.331,409.491,171.834,34.486,156.457
C05180=1054.409,197.083,409.515,171.832,34.483,156.456
C05181=1054.403,196.833,409.540,171.830,34.481,156.456
C05182=1054.397,196.586,409.564,171.827,34.478,156.455
C05183=1054.391,196.336,409.589,171.825,34.475,156.455
C05184=1054.385,196.087,409.613,171.823,34.473,156.454
C05185=1054.379,195.839,409.637,171.820,34.470,156.454
C05186=1054.373,195.589,409.661,171.818,34.467,156.453
C05187=1054.367,195.341,409.685,171.815,34.465,156.453
C05188=1054.361,195.092,409.710,171.813,34.461,156.452
C05189=1054.355,194.844,409.733,171.811,34.459,156.452
C05190=1054.349,194.594,409.758,171.809,34.456,156.451
C05191=1054.343,194.347,409.782,171.807,34.453,156.451
C05192=1054.337,194.097,409.807,171.803,34.451,156.450
C05193=1054.331,193.849,409.831,171.801,34.448,156.450
C05194=1054.325,193.600,409.855,171.799,34.445,156.449
C05195=1054.319,193.352,409.879,171.797,34.443,156.449
C05196=1054.313,193.102,409.904,171.795,34.440,156.448
C05197=1054.307,192.854,409.927,171.793,34.437,156.448
C05198=1054.301,192.605,409.952,171.790,34.435,156.447
C05199=1054.295,192.356,409.976,171.788,34.431,156.447
C05200=1054.290,192.108,410.000,171.785,34.429,156.446
C05201=1054.283,191.859,410.024,171.783,34.426,156.446
C05202=1054.278,191.610,410.048,171.781,34.423,156.445
C05203=1054.271,191.361,410.071,171.778,34.421,156.445
C05204=1054.266,191.112,410.096,171.776,34.418,156.444
C05205=1054.259,190.863,410.120,171.774,34.415,156.444
C05206=1054.253,190.580,410.147,171.772,34.412,156.443
C05207=1054.246,190.295,410.174,171.769,34.409,156.442
C05208=1054.240,190.012,410.203,171.766,34.406,156.442
C05209=1054.233,189.727,410.230,171.763,34.403,156.441
C05210=1054.227,189.478,410.254,171.761,34.400,156.441
C05211=1054.221,189.230,410.277,171.759,34.398,156.440
C05212=1054.215,188.981,410.302,171.757,34.395,156.440
C05213=1054.209,188.732,410.325,171.755,34.392,156.439
C05214=1054.204,188.483,410.350,171.753,34.390,156.439
C05215=1054.197,188.234,410.373,171.751,34.387,156.438
C05216=1054.192,187.986,410.397,171.747,34.384,156.438
C05217=1054.186,187.737,410.421,171.745,34.381,156.437
C05218=1054.181,187.488,410.445,171.743,34.379,156.437
C05219=1054.175,187.239,410.469,171.741,34.376,156.436
C05220=1054.169,186.990,410.493,171.739,34.373,156.436
C05221=1054.163,186.742,410.517,171.737,34.371,156.436
C05222=1054.158,186.493,410.541,171.735,34.368,156.435
C05223=1054.152,186.244,410.564,171.733,34.365,156.434
C05224=1054.145,185.995,410.588,171.731,34.363,156.434
C05225=1054.140,185.746,410.612,171.727,34.360,156.433
C05226=1054.134,185.498,410.635,171.725,34.357,156.433
C05227=1054.128,185.249,410.660,171.723,34.354,156.433
C05228=1054.122,185.000,410.684,171.721,34.352,156.432
C05229=1054.117,184.751,410.707,171.719,34.349,156.432
C05230=1054.111,184.503,410.731,171.717,34.346,156.431
C05231=1054.105,184.253,410.754,171.715,34.344,156.431
C05232=1054.099,184.005,410.778,171.713,34.341,156.430
C05233=1054.093,183.757,410.802,171.710,34.339,156.430
C05234=1054.086,183.507,410.825,171.708,34.336,156.429
C05235=1054.080,183.259,410.848,171.705,34.334,156.429
C05236=1054.074,183.009,410.872,171.703,34.331,156.428
C05237=1054.068,182.761,410.895,171.701,34.329,156.428
C05238=1054.062,182.512,410.918,171.699,34.326,156.427
C05239=1054.055,182.263,410.942,171.697,34.323,156.427
C05240=1054.050,182.014,410.965,171.695,34.321,156.426
C05241=1054.044,181.765,410.988,171.693,34.318,156.426
C05242=1054.037,181.516,411.012,171.691,34.316,156.426
C05243=1054.032,181.267,411.035,171.688,34.313,156.425
C05244=1054.026,181.019,411.059,171.685,34.310,156.425
C05245=1054.019,180.770,411.082,171.683,34.308,156.424
C05246=1054.013,180.521,411.106,171.681,34.306,156.424
C05247=1054.007,180.273,411.128,171.679,34.304,156.423
C05248=1054.001,180.024,411.151,171.677,34.301,156.423
C05249=1053.994,179.775,411.175,171.675,34.299,156.422
C05250=1053.989,179.526,411.198,171.673,34.296,156.422
C05251=1053.983,179.277,411.221,171.671,34.293,156.422
C05252=1053.976,179.028,411.245,171.669,34.291,156.421
C05253=1053.971,178.779,411.268,171.666,34.288,156.421
C05254=1053.965,178.530,411.291,171.664,34.286,156.420
C05255=1053.959,178.282,411.315,171.662,34.283,156.420
C05256=1053.952,178.032,411.338,171.659,34.281,156.419
C05257=1053.946,177.784,411.360,171.657,34.278,156.419
C05258=1053.940,177.535,411.384,171.655,34.276,156.418
C05259=1053.934,177.287,411.407,171.653,34.273,156.418
C05260=1053.928,177.037,411.430,171.651,34.271,156.418
C05261=1053.922,176.788,411.453,171.649,34.268,156.417
C05262=1053.916,176.540,411.477,171.647,34.266,156.417
C05263=1053.910,176.291,411.500,171.644,34.263,156.416
C05264=1053.905,176.042,411.523,171.642,34.261,156.416
C05265=1053.898,175.793,411.546,171.640,34.258,156.415
C05266=1053.891,175.544,411.569,171.638,34.256,156.415
C05267=1053.886,175.296,411.592,171.636,34.253,156.414
C05268=1053.880,175.047,411.615,171.634,34.251,156.414
C05269=1053.874,174.798,411.638,171.632,34.248,156.413
C05270=1053.867,174.513,411.665,171.630,34.245,156.413
C05271=1053.860,174.228,411.691,171.627,34.242,156.412
C05272=1053.853,173.944,411.717,171.625,34.239,156.412
C05273=1053.847,173.660,411.744,171.622,34.237,156.411
C05274=1053.841,173.411,411.766,171.620,34.234,156.411
C05275=1053.835,173.162,411.789,171.618,34.232,156.411
C05276=1053.829,172.913,411.812,171.616,34.229,156.410
C05277=1053.823,172.664,411.835,171.614,34.227,156.410
C05278=1053.817,172.415,411.858,171.612,34.224,156.409
C05279=1053.811,172.166,411.881,171.610,34.222,156.409
C05280=1053.805,171.918,411.904,171.608,34.219,156.408
C05281=1053.799,171.669,411.926,171.606,34.217,156.408
C05282=1053.793,171.420,411.950,171.604,34.214,156.407
C05283=1053.787,171.171,411.973,171.601,34.212,156.407
C05284=1053.782,170.923,411.996,171.599,34.209,156.406
C05285=1053.776,170.674,412.019,171.597,34.206,156.406
C05286=1053.769,170.424,412.042,171.595,34.204,156.406
C05287=1053.763,170.175,412.065,171.593,34.201,156.405
C05288=1053.757,169.927,412.088,171.591,34.199,156.405
C05289=1053.752,169.678,412.111,171.589,34.196,156.404
C05290=1053.746,169.429,412.133,171.587,34.194,156.404
C05291=1053.739,169.180,412.156,171.585,34.191,156.403
C05292=1053.734,168.931,412.178,171.583,34.189,156.403
C05293=1053.728,168.682,412.201,171.581,34.186,156.402
C05294=1053.723,168.433,412.224,171.578,34.184,156.402
C05295=1053.717,168.184,412.247,171.576,34.181,156.402
C05296=1053.710,167.935,412.269,171.574,34.179,156.401
C05297=1053.705,167.686,412.292,171.572,34.176,156.401
C05298=1053.699,167.438,412.315,171.570,34.174,156.400
C05299=1053.693,167.189,412.338,171.568,34.172,156.400
C05300=1053.687,166.940,412.361,171.566,34.169,156.399
C05301=1053.681,166.691,412.383,171.564,34.167,156.399
C05302=1053.676,166.442,412.406,171.562,34.164,156.398
C05303=1053.670,166.193,412.429,171.560,34.162,156.398
C05304=1053.664,165.944,412.452,171.558,34.159,156.398
C05305=1053.658,165.695,412.474,171.555,34.157,156.397
C05306=1053.652,165.446,412.497,171.553,34.154,156.397
C05307=1053.646,165.198,412.520,171.551,34.151,156.396
C05308=1053.641,164.949,412.542,171.549,34.149,156.396
C05309=1053.636,164.700,412.565,171.547,34.146,156.395
C05310=1053.629,164.451,412.587,171.546,34.144,156.395
C05311=1053.623,164.202,412.610,171.544,34.141,156.394
C05312=1053.618,163.953,412.632,171.542,34.139,156.394
C05313=1053.612,163.704,412.655,171.540,34.136,156.394
C05314=1053.606,163.455,412.677,171.538,34.134,156.393
C05315=1053.600,163.206,412.700,171.536,34.131,156.393
C05316=1053.595,162.957,412.723,171.533,34.129,156.392
C05317=1053.589,162.708,412.746,171.531,34.126,156.392
C05318=1053.582,162.459,412.768,171.529,34.124,156.391
C05319=1053.577,162.211,412.790,171.527,34.121,156.391
C05320=1053.572,161.962,412.813,171.525,34.119,156.390
C05321=1053.566,161.713,412.836,171.523,34.116,156.390
C05322=1053.560,161.464,412.858,171.521,34.114,156.389
C05323=1053.554,161.215,412.880,171.520,34.111,156.389
C05324=1053.548,160.966,412.903,171.518,34.109,156.389
C05325=1053.543,160.716,412.925,171.516,34.107,156.388
C05326=1053.537,160.468,412.948,171.514,34.104,156.388
C05327=1053.530,160.219,412.970,171.512,34.102,156.387
C05328=1053.525,159.970,412.992,171.509,34.099,156.387
C05329=1053.519,159.722,413.014,171.507,34.097,156.387
C05330=1053.513,159.473,413.036,171.505,34.095,156.386
C05331=1053.507,159.224,413.059,171.503,34.092,156.386
C05332=1053.501,158.974,413.080,171.501,34.089,156.385
C05333=1053.495,158.726,413.103,171.499,34.087,156.385
C05334=1053.488,158.440,413.128,171.497,34.084,156.384
C05335=1053.482,158.156,413.154,171.495,34.082,156.384
C05336=1053.474,157.870,413.179,171.493,34.079,156.383
C05337=1053.468,157.586,413.205,171.491,34.076,156.383
C05338=1053.461,157.337,413.227,171.489,34.074,156.382
C05339=1053.455,157.087,413.248,171.487,34.072,156.382
C05340=1053.450,156.839,413.271,171.485,34.069,156.382
C05341=1053.444,156.590,413.293,171.482,34.067,156.381
C05342=1053.437,156.341,413.315,171.480,34.064,156.381
C05343=1053.432,156.092,413.337,171.478,34.062,156.380
C05344=1053.426,155.843,413.360,171.476,34.060,156.380
C05345=1053.419,155.594,413.381,171.474,34.057,156.380
C05346=1053.414,155.345,413.403,171.473,34.055,156.379
C05347=1053.408,155.097,413.425,171.471,34.053,156.379
C05348=1053.402,154.847,413.447,171.469,34.050,156.378
C05349=1053.396,154.598,413.469,171.467,34.048,156.378
C05350=1053.390,154.349,413.492,171.465,34.045,156.377
C05351=1053.384,154.100,413.513,171.463,34.043,156.377
C05352=1053.378,153.851,413.535,171.461,34.041,156.377
C05353=1053.372,153.603,413.557,171.459,34.038,156.376
C05354=1053.366,153.354,413.579,171.457,34.036,156.376
C05355=1053.360,153.104,413.601,171.455,34.034,156.375
C05356=1053.354,152.855,413.622,171.453,34.031,156.375
C05357=1053.348,152.607,413.645,171.451,34.029,156.375
C05358=1053.342,152.358,413.666,171.449,34.027,156.374
C05359=1053.337,152.109,413.688,171.447,34.024,156.374
C05360=1053.330,151.859,413.710,171.445,34.021,156.373
C05361=1053.324,151.611,413.732,171.443,34.020,156.373
C05362=1053.318,151.362,413.754,171.442,34.017,156.373
C05363=1053.312,151.113,413.775,171.440,34.015,156.372
C05364=1053.307,150.863,413.797,171.438,34.013,156.372
C05365=1053.300,150.615,413.820,171.436,34.010,156.371
C05366=1053.294,150.366,413.841,171.434,34.007,156.371
C05367=1053.289,150.117,413.863,171.432,34.005,156.370
C05368=1053.282,149.868,413.884,171.430,34.003,156.370
C05369=1053.276,149.619,413.906,171.428,34.001,156.370
C05370=1053.271,149.369,413.928,171.426,33.998,156.369
C05371=1053.265,149.121,413.949,171.424,33.996,156.369
C05372=1053.259,148.872,413.972,171.422,33.993,156.368
C05373=1053.253,148.623,413.993,171.420,33.991,156.368
C05374=1053.247,148.374,414.015,171.418,33.989,156.368
C05375=1053.241,148.125,414.036,171.417,33.987,156.367
C05376=1053.235,147.876,414.058,171.415,33.984,156.367
C05377=1053.229,147.627,414.080,171.413,33.982,156.366
C05378=1053.222,147.378,414.101,171.411,33.979,156.366
C05379=1053.217,147.129,414.122,171.409,33.977,156.366
C05380=1053.211,146.880,414.144,171.407,33.975,156.365
C05381=1053.205,146.631,414.166,171.405,33.972,156.365
C05382=1053.199,146.382,414.187,171.404,33.971,156.364
C05383=1053.193,146.133,414.209,171.401,33.968,156.364
C05384=1053.187,145.884,414.230,171.399,33.965,156.364
C05385=1053.181,145.635,414.252,171.397,33.964,156.363
C05386=1053.175,145.386,414.273,171.395,33.961,156.363
C05387=1053.169,145.137,414.295,171.393,33.958,156.362
C05388=1053.163,144.888,414.316,171.392,33.957,156.362
C05389=1053.157,144.639,414.338,171.390,33.954,156.362
C05390=1053.151,144.390,414.359,171.388,33.952,156.361
C05391=1053.145,144.141,414.381,171.386,33.949,156.361
C05392=1053.139,143.892,414.403,171.384,33.947,156.360
C05393=1053.133,143.643,414.424,171.382,33.945,156.360
C05394=1053.126,143.394,414.445,171.381,33.942,156.360
C05395=1053.120,143.144,414.466,171.379,33.941,156.359
C05396=1053.115,142.896,414.487,171.377,33.938,156.359
C05397=1053.109,142.647,414.509,171.375,33.935,156.358
C05398=1053.102,142.362,414.534,171.373,33.933,156.358
C05399=1053.095,142.076,414.557,171.370,33.930,156.357
C05400=1053.088,141.791,414.582,171.368,33.928,156.357
C05401=1053.082,141.506,414.607,171.366,33.925,156.357
C05402=1053.075,141.256,414.628,171.364,33.923,156.356
C05403=1053.070,141.008,414.649,171.362,33.920,156.356
C05404=1053.064,140.759,414.670,171.361,33.918,156.355
C05405=1053.057,140.510,414.692,171.359,33.916,156.355
C05406=1053.052,140.261,414.713,171.357,33.914,156.355
C05407=1053.046,140.011,414.734,171.355,33.911,156.354
C05408=1053.040,139.763,414.756,171.353,33.909,156.354
C05409=1053.034,139.514,414.777,171.352,33.907,156.353
C05410=1053.027,139.265,414.798,171.350,33.904,156.353
C05411=1053.022,139.016,414.819,171.348,33.902,156.353
C05412=1053.016,138.766,414.840,171.346,33.900,156.352
C05413=1053.010,138.517,414.862,171.344,33.897,156.352
C05414=1053.003,138.269,414.883,171.343,33.895,156.351
C05415=1052.998,138.019,414.904,171.340,33.893,156.351
C05416=1052.992,137.771,414.925,171.338,33.891,156.351
C05417=1052.986,137.521,414.947,171.336,33.888,156.350
C05418=1052.980,137.273,414.967,171.334,33.886,156.350
C05419=1052.974,137.023,414.988,171.333,33.884,156.349
C05420=1052.968,136.774,415.010,171.331,33.882,156.349
C05421=1052.962,136.525,415.030,171.329,33.879,156.349
C05422=1052.955,136.276,415.051,171.327,33.877,156.348
C05423=1052.950,136.027,415.072,171.325,33.875,156.348
C05424=1052.943,135.778,415.093,171.324,33.872,156.347
C05425=1052.937,135.529,415.115,171.322,33.870,156.347
C05426=1052.932,135.280,415.135,171.320,33.868,156.347
C05427=1052.925,135.031,415.156,171.318,33.866,156.346
C05428=1052.920,134.782,415.177,171.317,33.863,156.346
C05429=1052.913,134.533,415.198,171.315,33.861,156.346
C05430=1052.907,134.284,415.219,171.313,33.859,156.345
C05431=1052.901,134.035,415.240,171.311,33.857,156.345
C05432=1052.896,133.786,415.261,171.310,33.854,156.344
C05433=1052.889,133.537,415.282,171.307,33.852,156.344
C05434=1052.884,133.288,415.303,171.305,33.850,156.344
C05435=1052.878,133.038,415.324,171.303,33.847,156.343
C05436=1052.871,132.790,415.344,171.301,33.845,156.343
C05437=1052.866,132.540,415.365,171.300,33.843,156.342
C05438=1052.860,132.292,415.387,171.298,33.841,156.342
C05439=1052.853,132.042,415.407,171.296,33.838,156.342
C05440=1052.848,131.794,415.428,171.294,33.836,156.341
C05441=1052.842,131.544,415.449,171.293,33.834,156.341
C05442=1052.836,131.296,415.470,171.291,33.832,156.340
C05443=1052.829,131.046,415.490,171.289,33.829,156.340
C05444=1052.824,130.797,415.511,171.287,33.827,156.340
C05445=1052.817,130.548,415.532,171.286,33.825,156.339
C05446=1052.812,130.299,415.552,171.284,33.823,156.339
C05447=1052.805,130.049,415.573,171.282,33.821,156.339
C05448=1052.799,129.801,415.593,171.280,33.818,156.338
C05449=1052.793,129.551,415.614,171.279,33.816,156.338
C05450=1052.786,129.303,415.635,171.277,33.814,156.337
C05451=1052.780,129.054,415.655,171.275,33.812,156.337
C05452=1052.774,128.804,415.676,171.273,33.809,156.337
C05453=1052.768,128.556,415.697,171.271,33.807,156.336
C05454=1052.761,128.306,415.717,171.269,33.806,156.336
C05455=1052.756,128.057,415.738,171.267,33.803,156.336
C05456=1052.750,127.808,415.758,171.265,33.801,156.335
C05457=1052.744,127.559,415.779,171.263,33.798,156.335
C05458=1052.738,127.310,415.799,171.262,33.797,156.334
